KUKA KRL program: ps_a_stb_res_co3.src, ps_a_stb_res_co3.dat

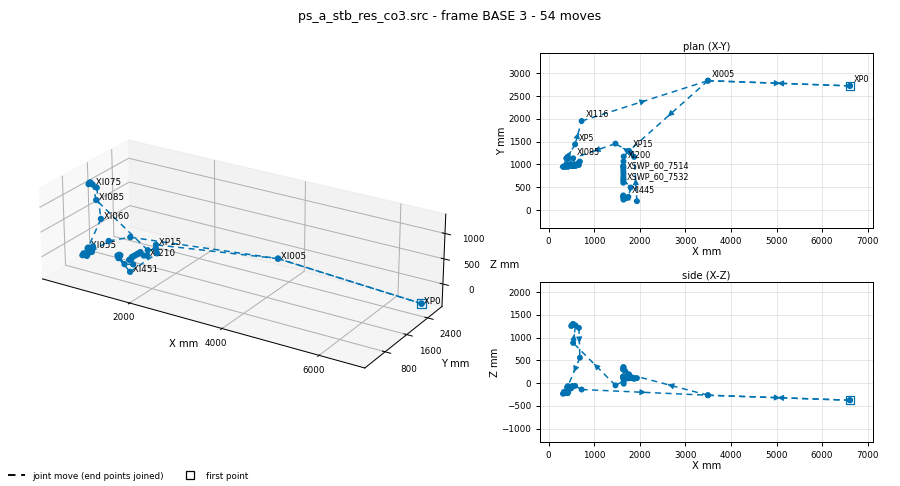
[picture p0: tool path of ps_a_stb_res_co3.src in frame BASE 3, 54 of 54 moves have a stored position in this frame; points joined in program order, loops and branches not executed]
--- ps_a_stb_res_co3.src ---
&ACCESS RVO1
&COMMENT Solda Atego ETB
&PARAM DISKPATH = KRC:\R1\Program\inpro_nao_mexer
DEF ps_a_stb_res_co3( )
;FOLD INI
;FOLD SPOTTECH INI
USERSPOT(#INIT)
;ENDFOLD (SPOTTECH INI)
;FOLD GRIPPERTECH INI
USER_GRP(0,DUMMY,DUMMY,GDEFAULT)
;ENDFOLD (GRIPPERTECH INI)
  ;FOLD USER INI
    ;Make your modifications here

  ;ENDFOLD (USER INI)
;ENDFOLD (INI)

; Caracterizacao dos meios de producao
; Changes: Solda Respot - ATEGO STB
; Versao Atual:05/01/2016
; Ferramenta: Gun C3
; Name: P13.050-R2
; optimised

chk_w4_wechs_ok( )      ; CHECK GUN C3

;FOLD PTP P0 Vel=100 % PDAT0 Tool[4]:Gun C3 Base[3]:Atego/Axor;%{PE}%R 8.2.20,%MKUKATPBASIS,%CMOVE,%VPTP,%P 1:PTP, 2:P0, 3:, 5:100, 7:PDAT0
$BWDSTART=FALSE
PDAT_ACT=PPDAT0
FDAT_ACT=FP0
BAS(#PTP_PARAMS,100)
PTP XP0
;ENDFOLD

if MaxStandMenge (3) then
 MaxStandmengeErreicht (3)
endif

IF (NOT(GHOST())) THEN
if FraesAnf (3) then
 e_fraes4 ( )
endif
ENDIF

;FOLD PTP l005 Vel=100 % P_OLP2 Tool[4]:Gun C3 Base[3]:Atego/Axor;%{PE}%R 8.2.20,%MKUKATPBASIS,%CMOVE,%VPTP,%P 1:PTP, 2:l005, 3:, 5:100, 7:P_OLP2
$BWDSTART=FALSE
PDAT_ACT=PP_OLP2
FDAT_ACT=Fl005
BAS(#PTP_PARAMS,100)
PTP Xl005
;ENDFOLD

; AGUARDA LIBERACAO PARA SOLDAR RESPOT
;FOLD OUT 3338 'R2 solda geometria Ok' State=FALSE ;%{PE}%R 8.2.20,%MKUKATPBASIS,%COUT,%VOUTX,%P 2:3338, 3:R2 solda geometria Ok, 5:FALSE, 6:
$OUT[3338]=FALSE
;ENDFOLD
;FOLD OUT 3348 'Fora area GEOBOX' State=FALSE ;%{PE}%R 8.2.20,%MKUKATPBASIS,%COUT,%VOUTX,%P 2:3348, 3:Fora area GEOBOX, 5:FALSE, 6:
$OUT[3348]=FALSE
;ENDFOLD
;FOLD OUT 3380 'Lib. p/ soldar Res Axor/Atego' State=TRUE ;%{PE}%R 8.2.20,%MKUKATPBASIS,%COUT,%VOUTX,%P 2:3380, 3:Lib. p/ soldar Res Axor/Atego, 5:TRUE, 6:
$OUT[3380]=TRUE
;ENDFOLD
;FOLD WAIT FOR ( IN 3380 'Lib. p/ soldar Res Axor/Atego' );%{PE}%R 8.2.20,%MKUKATPBASIS,%CEXT_WAIT_FOR,%VEXT_WAIT_FOR,%P 2:, 4:, 5:$IN, 6:3380, 7:Lib. p/ soldar Res Axor/Atego, 9:
WAIT FOR  ( $IN[3380] )
;ENDFOLD
;FOLD OUT 3380 'Lib. p/ soldar Res Axor/Atego' State=FALSE ;%{PE}%R 8.2.20,%MKUKATPBASIS,%COUT,%VOUTX,%P 2:3380, 3:Lib. p/ soldar Res Axor/Atego, 5:FALSE, 6:
$OUT[3380]=FALSE
;ENDFOLD

; LIGA INTERTRAVAMENTO 1 C/ R1
;FOLD Collision.Monitoring_1_On ;%{PE}%MKUKATPUSER
COLLSTOP( 1, 1 ) ;Interrupt-Controlled
;ENDFOLD

; LIGA INTERTRAVAMENTO 4 C/ R4
;FOLD Collision.Monitoring_4_On ;%{PE}%MKUKATPUSER
COLLSTOP( 4, 1 ) ;Interrupt-Controlled
;ENDFOLD

; LIGA INTERTRAVAMENTO 12 C/ R1
;FOLD Collision.Monitoring_AREA_6_On ;%{PE}%MKUKATPUSER
COLLSTOP( 12, 1 ) ;not Interrupt-Controlled
;ENDFOLD

;FOLD PTP P15 CONT Vel=100 % xlarge Tool[4]:Gun C3 Base[3]:Atego/Axor;%{PE}%R 8.2.20,%MKUKATPBASIS,%CMOVE,%VPTP,%P 1:PTP, 2:P15, 3:C_DIS, 5:100, 7:xlarge
$BWDSTART=FALSE
PDAT_ACT=Pxlarge
FDAT_ACT=FP15
BAS(#PTP_PARAMS,100)
PTP XP15 C_DIS
;ENDFOLD
;FOLD PTP l210 CONT Vel=100 % large Tool[4]:Gun C3 Base[3]:Atego/Axor;%{PE}%R 8.2.20,%MKUKATPBASIS,%CMOVE,%VPTP,%P 1:PTP, 2:l210, 3:C_DIS, 5:100, 7:large
$BWDSTART=FALSE
PDAT_ACT=Plarge
FDAT_ACT=Fl210
BAS(#PTP_PARAMS,100)
PTP Xl210 C_DIS
;ENDFOLD
;FOLD PTP l200 CONT Vel=100 % medium Tool[4]:Gun C3 Base[3]:Atego/Axor;%{PE}%R 8.2.20,%MKUKATPBASIS,%CMOVE,%VPTP,%P 1:PTP, 2:l200, 3:C_DIS, 5:100, 7:medium
$BWDSTART=FALSE
PDAT_ACT=Pmedium
FDAT_ACT=Fl200
BAS(#PTP_PARAMS,100)
PTP Xl200 C_DIS
;ENDFOLD
;FOLD PTP l195 CONT Vel=100 % fin Tool[4]:Gun C3 Base[3]:Atego/Axor;%{PE}%R 8.2.20,%MKUKATPBASIS,%CMOVE,%VPTP,%P 1:PTP, 2:l195, 3:C_DIS, 5:100, 7:fin
$BWDSTART=FALSE
PDAT_ACT=Pfin
FDAT_ACT=Fl195
BAS(#PTP_PARAMS,100)
PTP Xl195 C_DIS
;ENDFOLD

;FOLD ; SWP_60_7512;%{PE}%R 8.2.20,%MKUKATPBASIS,%CCOMMENT,%VNORMAL,%P 2:SWP_60_7512
;ENDFOLD
;FOLD PTP SWP_60_7512 vmax SPOT Gun=3 RETR CLS PgNo1=204 ACTIVE=1 Tool[4]:Gun C3 Base[3]:Atego/Axor;%{PE}%R 8.2.2,%MKUKATPSPOT,%CSPOT,%VPTP,%P 1:PTP, 2:SWP_60_7512, 3:, 5:100, 7:vmax, 10:3, 12:#FIRST, 14:#CLO, 16:204, 18:1, 20:0, 22:0, 24:1, 25:NORMAL
$BWDSTART=FALSE
PDAT_ACT=Pvmax
FDAT_ACT=FSWP_60_7512
BAS(#PTP_PARAMS,Pvmax.VEL)
S_ACT.GUN=3
S_ACT.PAIR=SDEFAULT.PAIR
S_ACT.RETR=#CLO
S_ACT.CLO_TM=1
S_ACT.PGNO1=204
S_ACT.PGNO2=SDEFAULT.PGNO2
S_ACT.PRESS1=SDEFAULT.PRESS1
S_ACT.PRESS2=SDEFAULT.PRESS2
S_READY=FALSE
PTP XSWP_60_7512
USERSPOT(#SPOT, S_ACT)
WAIT FOR S_READY
;ENDFOLD

;FOLD ; SWP_60_7510;%{PE}%R 8.2.20,%MKUKATPBASIS,%CCOMMENT,%VNORMAL,%P 2:SWP_60_7510
;ENDFOLD
;FOLD PTP SWP_60_7510 vmax SPOT Gun=3 RETR CLS PgNo1=204 ACTIVE=1 Tool[4]:Gun C3 Base[3]:Atego/Axor;%{PE}%R 8.2.2,%MKUKATPSPOT,%CSPOT,%VPTP,%P 1:PTP, 2:SWP_60_7510, 3:, 5:100, 7:vmax, 10:3, 12:#FIRST, 14:#CLO, 16:204, 18:1, 20:0, 22:0, 24:1, 25:NORMAL
$BWDSTART=FALSE
PDAT_ACT=Pvmax
FDAT_ACT=FSWP_60_7510
BAS(#PTP_PARAMS,Pvmax.VEL)
S_ACT.GUN=3
S_ACT.PAIR=SDEFAULT.PAIR
S_ACT.RETR=#CLO
S_ACT.CLO_TM=1
S_ACT.PGNO1=204
S_ACT.PGNO2=SDEFAULT.PGNO2
S_ACT.PRESS1=SDEFAULT.PRESS1
S_ACT.PRESS2=SDEFAULT.PRESS2
S_READY=FALSE
PTP XSWP_60_7510
USERSPOT(#SPOT, S_ACT)
WAIT FOR S_READY
;ENDFOLD

;FOLD ; SWP_60_7508;%{PE}%R 8.2.20,%MKUKATPBASIS,%CCOMMENT,%VNORMAL,%P 2:SWP_60_7508
;ENDFOLD
;FOLD PTP SWP_60_7508 vmax SPOT Gun=3 RETR CLS PgNo1=204 ACTIVE=1 Tool[4]:Gun C3 Base[3]:Atego/Axor;%{PE}%R 8.2.2,%MKUKATPSPOT,%CSPOT,%VPTP,%P 1:PTP, 2:SWP_60_7508, 3:, 5:100, 7:vmax, 10:3, 12:#FIRST, 14:#CLO, 16:204, 18:1, 20:0, 22:0, 24:1, 25:NORMAL
$BWDSTART=FALSE
PDAT_ACT=Pvmax
FDAT_ACT=FSWP_60_7508
BAS(#PTP_PARAMS,Pvmax.VEL)
S_ACT.GUN=3
S_ACT.PAIR=SDEFAULT.PAIR
S_ACT.RETR=#CLO
S_ACT.CLO_TM=1
S_ACT.PGNO1=204
S_ACT.PGNO2=SDEFAULT.PGNO2
S_ACT.PRESS1=SDEFAULT.PRESS1
S_ACT.PRESS2=SDEFAULT.PRESS2
S_READY=FALSE
PTP XSWP_60_7508
USERSPOT(#SPOT, S_ACT)
WAIT FOR S_READY
;ENDFOLD

;FOLD ; SWP_60_7514;%{PE}%R 8.2.20,%MKUKATPBASIS,%CCOMMENT,%VNORMAL,%P 2:SWP_60_7514
;ENDFOLD
;FOLD PTP SWP_60_7514 vmax SPOT Gun=3 RETR CLS PgNo1=204 ACTIVE=1 Tool[4]:Gun C3 Base[3]:Atego/Axor;%{PE}%R 8.2.2,%MKUKATPSPOT,%CSPOT,%VPTP,%P 1:PTP, 2:SWP_60_7514, 3:, 5:100, 7:vmax, 10:3, 12:#FIRST, 14:#CLO, 16:204, 18:1, 20:0, 22:0, 24:1, 25:NORMAL
$BWDSTART=FALSE
PDAT_ACT=Pvmax
FDAT_ACT=FSWP_60_7514
BAS(#PTP_PARAMS,Pvmax.VEL)
S_ACT.GUN=3
S_ACT.PAIR=SDEFAULT.PAIR
S_ACT.RETR=#CLO
S_ACT.CLO_TM=1
S_ACT.PGNO1=204
S_ACT.PGNO2=SDEFAULT.PGNO2
S_ACT.PRESS1=SDEFAULT.PRESS1
S_ACT.PRESS2=SDEFAULT.PRESS2
S_READY=FALSE
PTP XSWP_60_7514
USERSPOT(#SPOT, S_ACT)
WAIT FOR S_READY
;ENDFOLD

;FOLD ; SWP_60_7518;%{PE}%R 8.2.20,%MKUKATPBASIS,%CCOMMENT,%VNORMAL,%P 2:SWP_60_7518
;ENDFOLD
;FOLD PTP SWP_60_7518 vmax SPOT Gun=3 RETR CLS PgNo1=204 ACTIVE=1 Tool[4]:Gun C3 Base[3]:Atego/Axor;%{PE}%R 8.2.2,%MKUKATPSPOT,%CSPOT,%VPTP,%P 1:PTP, 2:SWP_60_7518, 3:, 5:100, 7:vmax, 10:3, 12:#FIRST, 14:#CLO, 16:204, 18:1, 20:0, 22:0, 24:1, 25:NORMAL
$BWDSTART=FALSE
PDAT_ACT=Pvmax
FDAT_ACT=FSWP_60_7518
BAS(#PTP_PARAMS,Pvmax.VEL)
S_ACT.GUN=3
S_ACT.PAIR=SDEFAULT.PAIR
S_ACT.RETR=#CLO
S_ACT.CLO_TM=1
S_ACT.PGNO1=204
S_ACT.PGNO2=SDEFAULT.PGNO2
S_ACT.PRESS1=SDEFAULT.PRESS1
S_ACT.PRESS2=SDEFAULT.PRESS2
S_READY=FALSE
PTP XSWP_60_7518
USERSPOT(#SPOT, S_ACT)
WAIT FOR S_READY
;ENDFOLD

;FOLD ; SWP_60_7522;%{PE}%R 8.2.20,%MKUKATPBASIS,%CCOMMENT,%VNORMAL,%P 2:SWP_60_7522
;ENDFOLD
;FOLD PTP SWP_60_7522 vmax SPOT Gun=3 RETR CLS PgNo1=204 ACTIVE=1 Tool[4]:Gun C3 Base[3]:Atego/Axor;%{PE}%R 8.2.2,%MKUKATPSPOT,%CSPOT,%VPTP,%P 1:PTP, 2:SWP_60_7522, 3:, 5:100, 7:vmax, 10:3, 12:#FIRST, 14:#CLO, 16:204, 18:1, 20:0, 22:0, 24:1, 25:NORMAL
$BWDSTART=FALSE
PDAT_ACT=Pvmax
FDAT_ACT=FSWP_60_7522
BAS(#PTP_PARAMS,Pvmax.VEL)
S_ACT.GUN=3
S_ACT.PAIR=SDEFAULT.PAIR
S_ACT.RETR=#CLO
S_ACT.CLO_TM=1
S_ACT.PGNO1=204
S_ACT.PGNO2=SDEFAULT.PGNO2
S_ACT.PRESS1=SDEFAULT.PRESS1
S_ACT.PRESS2=SDEFAULT.PRESS2
S_READY=FALSE
PTP XSWP_60_7522
USERSPOT(#SPOT, S_ACT)
WAIT FOR S_READY
;ENDFOLD

;FOLD ; SWP_60_7524;%{PE}%R 8.2.20,%MKUKATPBASIS,%CCOMMENT,%VNORMAL,%P 2:SWP_60_7524
;ENDFOLD
;FOLD PTP SWP_60_7524 vmax SPOT Gun=3 RETR CLS PgNo1=204 ACTIVE=1 Tool[4]:Gun C3 Base[3]:Atego/Axor;%{PE}%R 8.2.2,%MKUKATPSPOT,%CSPOT,%VPTP,%P 1:PTP, 2:SWP_60_7524, 3:, 5:100, 7:vmax, 10:3, 12:#FIRST, 14:#CLO, 16:204, 18:1, 20:0, 22:0, 24:1, 25:NORMAL
$BWDSTART=FALSE
PDAT_ACT=Pvmax
FDAT_ACT=FSWP_60_7524
BAS(#PTP_PARAMS,Pvmax.VEL)
S_ACT.GUN=3
S_ACT.PAIR=SDEFAULT.PAIR
S_ACT.RETR=#CLO
S_ACT.CLO_TM=1
S_ACT.PGNO1=204
S_ACT.PGNO2=SDEFAULT.PGNO2
S_ACT.PRESS1=SDEFAULT.PRESS1
S_ACT.PRESS2=SDEFAULT.PRESS2
S_READY=FALSE
PTP XSWP_60_7524
USERSPOT(#SPOT, S_ACT)
WAIT FOR S_READY
;ENDFOLD

;FOLD ; SWP_60_7532;%{PE}%R 8.2.20,%MKUKATPBASIS,%CCOMMENT,%VNORMAL,%P 2:SWP_60_7532
;ENDFOLD
;FOLD PTP SWP_60_7532 vmax SPOT Gun=3 RETR CLS PgNo1=204 ACTIVE=1 Tool[4]:Gun C3 Base[3]:Atego/Axor;%{PE}%R 8.2.2,%MKUKATPSPOT,%CSPOT,%VPTP,%P 1:PTP, 2:SWP_60_7532, 3:, 5:100, 7:vmax, 10:3, 12:#FIRST, 14:#CLO, 16:204, 18:1, 20:0, 22:0, 24:1, 25:NORMAL
$BWDSTART=FALSE
PDAT_ACT=Pvmax
FDAT_ACT=FSWP_60_7532
BAS(#PTP_PARAMS,Pvmax.VEL)
S_ACT.GUN=3
S_ACT.PAIR=SDEFAULT.PAIR
S_ACT.RETR=#CLO
S_ACT.CLO_TM=1
S_ACT.PGNO1=204
S_ACT.PGNO2=SDEFAULT.PGNO2
S_ACT.PRESS1=SDEFAULT.PRESS1
S_ACT.PRESS2=SDEFAULT.PRESS2
S_READY=FALSE
PTP XSWP_60_7532
USERSPOT(#SPOT, S_ACT)
WAIT FOR S_READY
;ENDFOLD

;FOLD PTP l100 CONT Vel=100 % fin Tool[4]:Gun C3 Base[3]:Atego/Axor;%{PE}%R 8.2.20,%MKUKATPBASIS,%CMOVE,%VPTP,%P 1:PTP, 2:l100, 3:C_DIS, 5:100, 7:fin
$BWDSTART=FALSE
PDAT_ACT=Pfin
FDAT_ACT=Fl100
BAS(#PTP_PARAMS,100)
PTP Xl100 C_DIS
;ENDFOLD
;FOLD PTP l101 CONT Vel=100 % small Tool[4]:Gun C3 Base[3]:Atego/Axor;%{PE}%R 8.2.20,%MKUKATPBASIS,%CMOVE,%VPTP,%P 1:PTP, 2:l101, 3:C_DIS, 5:100, 7:small
$BWDSTART=FALSE
PDAT_ACT=Psmall
FDAT_ACT=Fl101
BAS(#PTP_PARAMS,100)
PTP Xl101 C_DIS
;ENDFOLD
;FOLD PTP l445 CONT Vel=100 % small Tool[4]:Gun C3 Base[3]:Atego/Axor;%{PE}%R 8.2.20,%MKUKATPBASIS,%CMOVE,%VPTP,%P 1:PTP, 2:l445, 3:C_DIS, 5:100, 7:small
$BWDSTART=FALSE
PDAT_ACT=Psmall
FDAT_ACT=Fl445
BAS(#PTP_PARAMS,100)
PTP Xl445 C_DIS
;ENDFOLD
;FOLD PTP l446 CONT Vel=100 % fin Tool[4]:Gun C3 Base[3]:Atego/Axor;%{PE}%R 8.2.20,%MKUKATPBASIS,%CMOVE,%VPTP,%P 1:PTP, 2:l446, 3:C_DIS, 5:100, 7:fin
$BWDSTART=FALSE
PDAT_ACT=Pfin
FDAT_ACT=Fl446
BAS(#PTP_PARAMS,100)
PTP Xl446 C_DIS
;ENDFOLD

;FOLD ; SWP_60_7536;%{PE}%R 8.2.20,%MKUKATPBASIS,%CCOMMENT,%VNORMAL,%P 2:SWP_60_7536
;ENDFOLD
;FOLD PTP SWP_60_7537 vmax SPOT Gun=3 RETR CLS PgNo1=204 ACTIVE=1 Tool[4]:Gun C3 Base[3]:Atego/Axor;%{PE}%R 8.2.2,%MKUKATPSPOT,%CSPOT,%VPTP,%P 1:PTP, 2:SWP_60_7537, 3:, 5:100, 7:vmax, 10:3, 12:#FIRST, 14:#CLO, 16:204, 18:1, 20:0, 22:0, 24:1, 25:NORMAL
$BWDSTART=FALSE
PDAT_ACT=Pvmax
FDAT_ACT=FSWP_60_7537
BAS(#PTP_PARAMS,Pvmax.VEL)
S_ACT.GUN=3
S_ACT.PAIR=SDEFAULT.PAIR
S_ACT.RETR=#CLO
S_ACT.CLO_TM=1
S_ACT.PGNO1=204
S_ACT.PGNO2=SDEFAULT.PGNO2
S_ACT.PRESS1=SDEFAULT.PRESS1
S_ACT.PRESS2=SDEFAULT.PRESS2
S_READY=FALSE
PTP XSWP_60_7537
USERSPOT(#SPOT, S_ACT)
WAIT FOR S_READY
;ENDFOLD

;FOLD ; SWP_60_7538;%{PE}%R 8.2.20,%MKUKATPBASIS,%CCOMMENT,%VNORMAL,%P 2:SWP_60_7538
;ENDFOLD
;FOLD PTP SWP_60_7538 vmax SPOT Gun=3 RETR CLS PgNo1=204 ACTIVE=1 Tool[4]:Gun C3 Base[3]:Atego/Axor;%{PE}%R 8.2.2,%MKUKATPSPOT,%CSPOT,%VPTP,%P 1:PTP, 2:SWP_60_7538, 3:, 5:100, 7:vmax, 10:3, 12:#FIRST, 14:#CLO, 16:204, 18:1, 20:0, 22:0, 24:1, 25:NORMAL
$BWDSTART=FALSE
PDAT_ACT=Pvmax
FDAT_ACT=FSWP_60_7538
BAS(#PTP_PARAMS,Pvmax.VEL)
S_ACT.GUN=3
S_ACT.PAIR=SDEFAULT.PAIR
S_ACT.RETR=#CLO
S_ACT.CLO_TM=1
S_ACT.PGNO1=204
S_ACT.PGNO2=SDEFAULT.PGNO2
S_ACT.PRESS1=SDEFAULT.PRESS1
S_ACT.PRESS2=SDEFAULT.PRESS2
S_READY=FALSE
PTP XSWP_60_7538
USERSPOT(#SPOT, S_ACT)
WAIT FOR S_READY
;ENDFOLD

;FOLD ; SWP_60_7540;%{PE}%R 8.2.20,%MKUKATPBASIS,%CCOMMENT,%VNORMAL,%P 2:SWP_60_7540
;ENDFOLD
;FOLD PTP SWP_60_7540 vmax SPOT Gun=3 RETR CLS PgNo1=204 ACTIVE=1 Tool[4]:Gun C3 Base[3]:Atego/Axor;%{PE}%R 8.2.2,%MKUKATPSPOT,%CSPOT,%VPTP,%P 1:PTP, 2:SWP_60_7540, 3:, 5:100, 7:vmax, 10:3, 12:#FIRST, 14:#CLO, 16:204, 18:1, 20:0, 22:0, 24:1, 25:NORMAL
$BWDSTART=FALSE
PDAT_ACT=Pvmax
FDAT_ACT=FSWP_60_7540
BAS(#PTP_PARAMS,Pvmax.VEL)
S_ACT.GUN=3
S_ACT.PAIR=SDEFAULT.PAIR
S_ACT.RETR=#CLO
S_ACT.CLO_TM=1
S_ACT.PGNO1=204
S_ACT.PGNO2=SDEFAULT.PGNO2
S_ACT.PRESS1=SDEFAULT.PRESS1
S_ACT.PRESS2=SDEFAULT.PRESS2
S_READY=FALSE
PTP XSWP_60_7540
USERSPOT(#SPOT, S_ACT)
WAIT FOR S_READY
;ENDFOLD

; LIGA INTERTRAVAMENTO 14 C/ R5
;FOLD Collision.Monitoring_AREA_8_On ;%{PE}%MKUKATPUSER
COLLSTOP( 14, 1 ) ;not Interrupt-Controlled
;ENDFOLD

;FOLD PTP l447 CONT Vel=100 % fin Tool[4]:Gun C3 Base[3]:Atego/Axor;%{PE}%R 8.2.20,%MKUKATPBASIS,%CMOVE,%VPTP,%P 1:PTP, 2:l447, 3:C_DIS, 5:100, 7:fin
$BWDSTART=FALSE
PDAT_ACT=Pfin
FDAT_ACT=Fl447
BAS(#PTP_PARAMS,100)
PTP Xl447 C_DIS
;ENDFOLD
;FOLD PTP l451 CONT Vel=100 % medium Tool[4]:Gun C3 Base[3]:Atego/Axor;%{PE}%R 8.2.20,%MKUKATPBASIS,%CMOVE,%VPTP,%P 1:PTP, 2:l451, 3:C_DIS, 5:100, 7:medium
$BWDSTART=FALSE
PDAT_ACT=Pmedium
FDAT_ACT=Fl451
BAS(#PTP_PARAMS,100)
PTP Xl451 C_DIS
;ENDFOLD
;FOLD PTP l103 CONT Vel=100 % medium Tool[4]:Gun C3 Base[3]:Atego/Axor;%{PE}%R 8.2.20,%MKUKATPBASIS,%CMOVE,%VPTP,%P 1:PTP, 2:l103, 3:C_DIS, 5:100, 7:medium
$BWDSTART=FALSE
PDAT_ACT=Pmedium
FDAT_ACT=Fl103
BAS(#PTP_PARAMS,100)
PTP Xl103 C_DIS
;ENDFOLD
;FOLD PTP l090 CONT Vel=100 % xlarge Tool[4]:Gun C3 Base[3]:Atego/Axor;%{PE}%R 8.2.20,%MKUKATPBASIS,%CMOVE,%VPTP,%P 1:PTP, 2:l090, 3:C_DIS, 5:100, 7:xlarge
$BWDSTART=FALSE
PDAT_ACT=Pxlarge
FDAT_ACT=Fl090
BAS(#PTP_PARAMS,100)
PTP Xl090 C_DIS
;ENDFOLD
;FOLD PTP l091 CONT Vel=100 % xlarge Tool[4]:Gun C3 Base[3]:Atego/Axor;%{PE}%R 8.2.20,%MKUKATPBASIS,%CMOVE,%VPTP,%P 1:PTP, 2:l091, 3:C_DIS, 5:100, 7:xlarge
$BWDSTART=FALSE
PDAT_ACT=Pxlarge
FDAT_ACT=Fl091
BAS(#PTP_PARAMS,100)
PTP Xl091 C_DIS
;ENDFOLD
;FOLD PTP l085 CONT Vel=100 % large Tool[4]:Gun C3 Base[3]:Atego/Axor;%{PE}%R 8.2.20,%MKUKATPBASIS,%CMOVE,%VPTP,%P 1:PTP, 2:l085, 3:C_DIS, 5:100, 7:large
$BWDSTART=FALSE
PDAT_ACT=Plarge
FDAT_ACT=Fl085
BAS(#PTP_PARAMS,100)
PTP Xl085 C_DIS
;ENDFOLD
;FOLD PTP l075 CONT Vel=100 % fin Tool[4]:Gun C3 Base[3]:Atego/Axor;%{PE}%R 8.2.20,%MKUKATPBASIS,%CMOVE,%VPTP,%P 1:PTP, 2:l075, 3:C_DIS, 5:100, 7:fin
$BWDSTART=FALSE
PDAT_ACT=Pfin
FDAT_ACT=Fl075
BAS(#PTP_PARAMS,100)
PTP Xl075 C_DIS
;ENDFOLD

;FOLD ; SWP_60_7784;%{PE}%R 8.2.20,%MKUKATPBASIS,%CCOMMENT,%VNORMAL,%P 2:SWP_60_7784
;ENDFOLD
;FOLD PTP SWP_60_7784 vmax SPOT Gun=3 RETR CLS PgNo1=201 ACTIVE=1 Tool[4]:Gun C3 Base[3]:Atego/Axor;%{PE}%R 8.2.2,%MKUKATPSPOT,%CSPOT,%VPTP,%P 1:PTP, 2:SWP_60_7784, 3:, 5:100, 7:vmax, 10:3, 12:#FIRST, 14:#CLO, 16:201, 18:1, 20:0, 22:0, 24:1, 25:NORMAL
$BWDSTART=FALSE
PDAT_ACT=Pvmax
FDAT_ACT=FSWP_60_7784
BAS(#PTP_PARAMS,Pvmax.VEL)
S_ACT.GUN=3
S_ACT.PAIR=SDEFAULT.PAIR
S_ACT.RETR=#CLO
S_ACT.CLO_TM=1
S_ACT.PGNO1=201
S_ACT.PGNO2=SDEFAULT.PGNO2
S_ACT.PRESS1=SDEFAULT.PRESS1
S_ACT.PRESS2=SDEFAULT.PRESS2
S_READY=FALSE
PTP XSWP_60_7784
USERSPOT(#SPOT, S_ACT)
WAIT FOR S_READY
;ENDFOLD

; DESLIGA INTERTRAVAMENTO 12 C/ R1
;FOLD Collision.Monitoring_AREA_6_Off . ;%{PE}%MKUKATPUSER
COLLSTOP( 12, 2+0 )
;ENDFOLD

;FOLD ; SWP_60_7782;%{PE}%R 8.2.20,%MKUKATPBASIS,%CCOMMENT,%VNORMAL,%P 2:SWP_60_7782
;ENDFOLD
;FOLD PTP SWP_60_7782 vmax SPOT Gun=3 RETR CLS PgNo1=201 ACTIVE=1 Tool[4]:Gun C3 Base[3]:Atego/Axor;%{PE}%R 8.2.2,%MKUKATPSPOT,%CSPOT,%VPTP,%P 1:PTP, 2:SWP_60_7782, 3:, 5:100, 7:vmax, 10:3, 12:#FIRST, 14:#CLO, 16:201, 18:1, 20:0, 22:0, 24:1, 25:NORMAL
$BWDSTART=FALSE
PDAT_ACT=Pvmax
FDAT_ACT=FSWP_60_7782
BAS(#PTP_PARAMS,Pvmax.VEL)
S_ACT.GUN=3
S_ACT.PAIR=SDEFAULT.PAIR
S_ACT.RETR=#CLO
S_ACT.CLO_TM=1
S_ACT.PGNO1=201
S_ACT.PGNO2=SDEFAULT.PGNO2
S_ACT.PRESS1=SDEFAULT.PRESS1
S_ACT.PRESS2=SDEFAULT.PRESS2
S_READY=FALSE
PTP XSWP_60_7782
USERSPOT(#SPOT, S_ACT)
WAIT FOR S_READY
;ENDFOLD

;FOLD ; SWP_60_7780;%{PE}%R 8.2.20,%MKUKATPBASIS,%CCOMMENT,%VNORMAL,%P 2:SWP_60_7780
;ENDFOLD
;FOLD PTP SWP_60_7780 vmax SPOT Gun=3 RETR CLS PgNo1=201 ACTIVE=1 Tool[4]:Gun C3 Base[3]:Atego/Axor;%{PE}%R 8.2.2,%MKUKATPSPOT,%CSPOT,%VPTP,%P 1:PTP, 2:SWP_60_7780, 3:, 5:100, 7:vmax, 10:3, 12:#FIRST, 14:#CLO, 16:201, 18:1, 20:0, 22:0, 24:1, 25:NORMAL
$BWDSTART=FALSE
PDAT_ACT=Pvmax
FDAT_ACT=FSWP_60_7780
BAS(#PTP_PARAMS,Pvmax.VEL)
S_ACT.GUN=3
S_ACT.PAIR=SDEFAULT.PAIR
S_ACT.RETR=#CLO
S_ACT.CLO_TM=1
S_ACT.PGNO1=201
S_ACT.PGNO2=SDEFAULT.PGNO2
S_ACT.PRESS1=SDEFAULT.PRESS1
S_ACT.PRESS2=SDEFAULT.PRESS2
S_READY=FALSE
PTP XSWP_60_7780
USERSPOT(#SPOT, S_ACT)
WAIT FOR S_READY
;ENDFOLD

;FOLD PTP l070 CONT Vel=100 % small Tool[4]:Gun C3 Base[3]:Atego/Axor;%{PE}%R 8.2.20,%MKUKATPBASIS,%CMOVE,%VPTP,%P 1:PTP, 2:l070, 3:C_DIS, 5:100, 7:small
$BWDSTART=FALSE
PDAT_ACT=Psmall
FDAT_ACT=Fl070
BAS(#PTP_PARAMS,100)
PTP Xl070 C_DIS
;ENDFOLD
;FOLD PTP l060 Vel=100 % P_OLP13 Tool[4]:Gun C3 Base[3]:Atego/Axor;%{PE}%R 8.2.20,%MKUKATPBASIS,%CMOVE,%VPTP,%P 1:PTP, 2:l060, 3:, 5:100, 7:P_OLP13
$BWDSTART=FALSE
PDAT_ACT=PP_OLP13
FDAT_ACT=Fl060
BAS(#PTP_PARAMS,100)
PTP Xl060
;ENDFOLD

; DESLIGA INTERTRAVAMENTO 14 C/ R5
;FOLD Collision.Monitoring_AREA_8_Off . ;%{PE}%MKUKATPUSER
COLLSTOP( 14, 2+0 )
;ENDFOLD

; LIGA INTERTRAVAMENTO 13 C/ R5
;FOLD Collision.Monitoring_AREA_7_On ;%{PE}%MKUKATPUSER
COLLSTOP( 13, 1 ) ;not Interrupt-Controlled
;ENDFOLD

;FOLD PTP l055 CONT Vel=100 % fin Tool[4]:Gun C3 Base[3]:Atego/Axor;%{PE}%R 8.2.20,%MKUKATPBASIS,%CMOVE,%VPTP,%P 1:PTP, 2:l055, 3:C_DIS, 5:100, 7:fin
$BWDSTART=FALSE
PDAT_ACT=Pfin
FDAT_ACT=Fl055
BAS(#PTP_PARAMS,100)
PTP Xl055 C_DIS
;ENDFOLD

;FOLD ; SWP_60_9076;%{PE}%R 8.2.20,%MKUKATPBASIS,%CCOMMENT,%VNORMAL,%P 2:SWP_60_9076
;ENDFOLD
;FOLD PTP SWP_60_9076 vmax SPOT Gun=3 RETR CLS PgNo1=202 ACTIVE=1 Tool[4]:Gun C3 Base[3]:Atego/Axor;%{PE}%R 8.2.2,%MKUKATPSPOT,%CSPOT,%VPTP,%P 1:PTP, 2:SWP_60_9076, 3:, 5:100, 7:vmax, 10:3, 12:#FIRST, 14:#CLO, 16:202, 18:1, 20:0, 22:0, 24:1, 25:NORMAL
$BWDSTART=FALSE
PDAT_ACT=Pvmax
FDAT_ACT=FSWP_60_9076
BAS(#PTP_PARAMS,Pvmax.VEL)
S_ACT.GUN=3
S_ACT.PAIR=SDEFAULT.PAIR
S_ACT.RETR=#CLO
S_ACT.CLO_TM=1
S_ACT.PGNO1=202
S_ACT.PGNO2=SDEFAULT.PGNO2
S_ACT.PRESS1=SDEFAULT.PRESS1
S_ACT.PRESS2=SDEFAULT.PRESS2
S_READY=FALSE
PTP XSWP_60_9076
USERSPOT(#SPOT, S_ACT)
WAIT FOR S_READY
;ENDFOLD

;FOLD ; SWP_60_9074;%{PE}%R 8.2.20,%MKUKATPBASIS,%CCOMMENT,%VNORMAL,%P 2:SWP_60_9074
;ENDFOLD
;FOLD PTP SWP_60_9074 vmax SPOT Gun=3 RETR CLS PgNo1=202 ACTIVE=1 Tool[4]:Gun C3 Base[3]:Atego/Axor;%{PE}%R 8.2.2,%MKUKATPSPOT,%CSPOT,%VPTP,%P 1:PTP, 2:SWP_60_9074, 3:, 5:100, 7:vmax, 10:3, 12:#FIRST, 14:#CLO, 16:202, 18:1, 20:0, 22:0, 24:1, 25:NORMAL
$BWDSTART=FALSE
PDAT_ACT=Pvmax
FDAT_ACT=FSWP_60_9074
BAS(#PTP_PARAMS,Pvmax.VEL)
S_ACT.GUN=3
S_ACT.PAIR=SDEFAULT.PAIR
S_ACT.RETR=#CLO
S_ACT.CLO_TM=1
S_ACT.PGNO1=202
S_ACT.PGNO2=SDEFAULT.PGNO2
S_ACT.PRESS1=SDEFAULT.PRESS1
S_ACT.PRESS2=SDEFAULT.PRESS2
S_READY=FALSE
PTP XSWP_60_9074
USERSPOT(#SPOT, S_ACT)
WAIT FOR S_READY
;ENDFOLD

;FOLD ; SWP_60_9072;%{PE}%R 8.2.20,%MKUKATPBASIS,%CCOMMENT,%VNORMAL,%P 2:SWP_60_9072
;ENDFOLD
;FOLD PTP SWP_60_9072 vmax SPOT Gun=3 RETR CLS PgNo1=202 ACTIVE=1 Tool[4]:Gun C3 Base[3]:Atego/Axor;%{PE}%R 8.2.2,%MKUKATPSPOT,%CSPOT,%VPTP,%P 1:PTP, 2:SWP_60_9072, 3:, 5:100, 7:vmax, 10:3, 12:#FIRST, 14:#CLO, 16:202, 18:1, 20:0, 22:0, 24:1, 25:NORMAL
$BWDSTART=FALSE
PDAT_ACT=Pvmax
FDAT_ACT=FSWP_60_9072
BAS(#PTP_PARAMS,Pvmax.VEL)
S_ACT.GUN=3
S_ACT.PAIR=SDEFAULT.PAIR
S_ACT.RETR=#CLO
S_ACT.CLO_TM=1
S_ACT.PGNO1=202
S_ACT.PGNO2=SDEFAULT.PGNO2
S_ACT.PRESS1=SDEFAULT.PRESS1
S_ACT.PRESS2=SDEFAULT.PRESS2
S_READY=FALSE
PTP XSWP_60_9072
USERSPOT(#SPOT, S_ACT)
WAIT FOR S_READY
;ENDFOLD

;FOLD ; SWP_60_9070;%{PE}%R 8.2.20,%MKUKATPBASIS,%CCOMMENT,%VNORMAL,%P 2:SWP_60_9070
;ENDFOLD
;FOLD PTP SWP_60_9070 vmax SPOT Gun=3 RETR CLS PgNo1=202 ACTIVE=1 Tool[4]:Gun C3 Base[3]:Atego/Axor;%{PE}%R 8.2.2,%MKUKATPSPOT,%CSPOT,%VPTP,%P 1:PTP, 2:SWP_60_9070, 3:, 5:100, 7:vmax, 10:3, 12:#FIRST, 14:#CLO, 16:202, 18:1, 20:0, 22:0, 24:1, 25:NORMAL
$BWDSTART=FALSE
PDAT_ACT=Pvmax
FDAT_ACT=FSWP_60_9070
BAS(#PTP_PARAMS,Pvmax.VEL)
S_ACT.GUN=3
S_ACT.PAIR=SDEFAULT.PAIR
S_ACT.RETR=#CLO
S_ACT.CLO_TM=1
S_ACT.PGNO1=202
S_ACT.PGNO2=SDEFAULT.PGNO2
S_ACT.PRESS1=SDEFAULT.PRESS1
S_ACT.PRESS2=SDEFAULT.PRESS2
S_READY=FALSE
PTP XSWP_60_9070
USERSPOT(#SPOT, S_ACT)
WAIT FOR S_READY
;ENDFOLD

;FOLD PTP l050 CONT Vel=100 % fin Tool[4]:Gun C3 Base[3]:Atego/Axor;%{PE}%R 8.2.20,%MKUKATPBASIS,%CMOVE,%VPTP,%P 1:PTP, 2:l050, 3:C_DIS, 5:100, 7:fin
$BWDSTART=FALSE
PDAT_ACT=Pfin
FDAT_ACT=Fl050
BAS(#PTP_PARAMS,100)
PTP Xl050 C_DIS
;ENDFOLD
;FOLD PTP l040 CONT Vel=100 % xlarge Tool[4]:Gun C3 Base[3]:Atego/Axor;%{PE}%R 8.2.20,%MKUKATPBASIS,%CMOVE,%VPTP,%P 1:PTP, 2:l040, 3:C_DIS, 5:100, 7:xlarge
$BWDSTART=FALSE
PDAT_ACT=Pxlarge
FDAT_ACT=Fl040
BAS(#PTP_PARAMS,100)
PTP Xl040 C_DIS
;ENDFOLD
;FOLD PTP l035 CONT Vel=100 % medium Tool[4]:Gun C3 Base[3]:Atego/Axor;%{PE}%R 8.2.20,%MKUKATPBASIS,%CMOVE,%VPTP,%P 1:PTP, 2:l035, 3:C_DIS, 5:100, 7:medium
$BWDSTART=FALSE
PDAT_ACT=Pmedium
FDAT_ACT=Fl035
BAS(#PTP_PARAMS,100)
PTP Xl035 C_DIS
;ENDFOLD
;FOLD PTP l025 CONT Vel=100 % fin Tool[4]:Gun C3 Base[3]:Atego/Axor;%{PE}%R 8.2.20,%MKUKATPBASIS,%CMOVE,%VPTP,%P 1:PTP, 2:l025, 3:C_DIS, 5:100, 7:fin
$BWDSTART=FALSE
PDAT_ACT=Pfin
FDAT_ACT=Fl025
BAS(#PTP_PARAMS,100)
PTP Xl025 C_DIS
;ENDFOLD

;FOLD ; SWP_60_9054;%{PE}%R 8.2.20,%MKUKATPBASIS,%CCOMMENT,%VNORMAL,%P 2:SWP_60_9054
;ENDFOLD
;FOLD PTP SWP_60_9054 vmax SPOT Gun=3 RETR CLS PgNo1=203 ACTIVE=1 Tool[4]:Gun C3 Base[3]:Atego/Axor;%{PE}%R 8.2.2,%MKUKATPSPOT,%CSPOT,%VPTP,%P 1:PTP, 2:SWP_60_9054, 3:, 5:100, 7:vmax, 10:3, 12:#FIRST, 14:#CLO, 16:203, 18:1, 20:0, 22:0, 24:1, 25:NORMAL
$BWDSTART=FALSE
PDAT_ACT=Pvmax
FDAT_ACT=FSWP_60_9054
BAS(#PTP_PARAMS,Pvmax.VEL)
S_ACT.GUN=3
S_ACT.PAIR=SDEFAULT.PAIR
S_ACT.RETR=#CLO
S_ACT.CLO_TM=1
S_ACT.PGNO1=203
S_ACT.PGNO2=SDEFAULT.PGNO2
S_ACT.PRESS1=SDEFAULT.PRESS1
S_ACT.PRESS2=SDEFAULT.PRESS2
S_READY=FALSE
PTP XSWP_60_9054
USERSPOT(#SPOT, S_ACT)
WAIT FOR S_READY
;ENDFOLD

;FOLD ; SWP_60_9048;%{PE}%R 8.2.20,%MKUKATPBASIS,%CCOMMENT,%VNORMAL,%P 2:SWP_60_9048
;ENDFOLD
;FOLD PTP SWP_60_9048 vmax SPOT Gun=3 RETR CLS PgNo1=203 ACTIVE=1 Tool[4]:Gun C3 Base[3]:Atego/Axor;%{PE}%R 8.2.2,%MKUKATPSPOT,%CSPOT,%VPTP,%P 1:PTP, 2:SWP_60_9048, 3:, 5:100, 7:vmax, 10:3, 12:#FIRST, 14:#CLO, 16:203, 18:1, 20:0, 22:0, 24:1, 25:NORMAL
$BWDSTART=FALSE
PDAT_ACT=Pvmax
FDAT_ACT=FSWP_60_9048
BAS(#PTP_PARAMS,Pvmax.VEL)
S_ACT.GUN=3
S_ACT.PAIR=SDEFAULT.PAIR
S_ACT.RETR=#CLO
S_ACT.CLO_TM=1
S_ACT.PGNO1=203
S_ACT.PGNO2=SDEFAULT.PGNO2
S_ACT.PRESS1=SDEFAULT.PRESS1
S_ACT.PRESS2=SDEFAULT.PRESS2
S_READY=FALSE
PTP XSWP_60_9048
USERSPOT(#SPOT, S_ACT)
WAIT FOR S_READY
;ENDFOLD

;FOLD ; SWP_60_9050;%{PE}%R 8.2.20,%MKUKATPBASIS,%CCOMMENT,%VNORMAL,%P 2:SWP_60_9050
;ENDFOLD
;FOLD PTP SWP_60_9050 vmax SPOT Gun=3 RETR CLS PgNo1=203 ACTIVE=1 Tool[4]:Gun C3 Base[3]:Atego/Axor;%{PE}%R 8.2.2,%MKUKATPSPOT,%CSPOT,%VPTP,%P 1:PTP, 2:SWP_60_9050, 3:, 5:100, 7:vmax, 10:3, 12:#FIRST, 14:#CLO, 16:203, 18:1, 20:0, 22:0, 24:1, 25:NORMAL
$BWDSTART=FALSE
PDAT_ACT=Pvmax
FDAT_ACT=FSWP_60_9050
BAS(#PTP_PARAMS,Pvmax.VEL)
S_ACT.GUN=3
S_ACT.PAIR=SDEFAULT.PAIR
S_ACT.RETR=#CLO
S_ACT.CLO_TM=1
S_ACT.PGNO1=203
S_ACT.PGNO2=SDEFAULT.PGNO2
S_ACT.PRESS1=SDEFAULT.PRESS1
S_ACT.PRESS2=SDEFAULT.PRESS2
S_READY=FALSE
PTP XSWP_60_9050
USERSPOT(#SPOT, S_ACT)
WAIT FOR S_READY
;ENDFOLD

;FOLD PTP P1 CONT Vel=100 % fin Tool[4]:Gun C3 Base[3]:Atego/Axor;%{PE}%R 8.2.20,%MKUKATPBASIS,%CMOVE,%VPTP,%P 1:PTP, 2:P1, 3:C_DIS, 5:100, 7:fin
$BWDSTART=FALSE
PDAT_ACT=Pfin
FDAT_ACT=FP1
BAS(#PTP_PARAMS,100)
PTP XP1 C_DIS
;ENDFOLD

;FOLD ; SWP_60_9052;%{PE}%R 8.2.20,%MKUKATPBASIS,%CCOMMENT,%VNORMAL,%P 2:SWP_60_9052
;ENDFOLD
;FOLD PTP SWP_60_9052 vmax SPOT Gun=3 RETR CLS PgNo1=203 ACTIVE=1 Tool[4]:Gun C3 Base[3]:Atego/Axor;%{PE}%R 8.2.2,%MKUKATPSPOT,%CSPOT,%VPTP,%P 1:PTP, 2:SWP_60_9052, 3:, 5:100, 7:vmax, 10:3, 12:#FIRST, 14:#CLO, 16:203, 18:1, 20:0, 22:0, 24:1, 25:NORMAL
$BWDSTART=FALSE
PDAT_ACT=Pvmax
FDAT_ACT=FSWP_60_9052
BAS(#PTP_PARAMS,Pvmax.VEL)
S_ACT.GUN=3
S_ACT.PAIR=SDEFAULT.PAIR
S_ACT.RETR=#CLO
S_ACT.CLO_TM=1
S_ACT.PGNO1=203
S_ACT.PGNO2=SDEFAULT.PGNO2
S_ACT.PRESS1=SDEFAULT.PRESS1
S_ACT.PRESS2=SDEFAULT.PRESS2
S_READY=FALSE
PTP XSWP_60_9052
USERSPOT(#SPOT, S_ACT)
WAIT FOR S_READY
;ENDFOLD

;FOLD PTP l020 CONT Vel=100 % fin Tool[4]:Gun C3 Base[3]:Atego/Axor;%{PE}%R 8.2.20,%MKUKATPBASIS,%CMOVE,%VPTP,%P 1:PTP, 2:l020, 3:C_DIS, 5:100, 7:fin
$BWDSTART=FALSE
PDAT_ACT=Pfin
FDAT_ACT=Fl020
BAS(#PTP_PARAMS,100)
PTP Xl020 C_DIS
;ENDFOLD
;FOLD PTP l010 CONT Vel=100 % medium Tool[4]:Gun C3 Base[3]:Atego/Axor;%{PE}%R 8.2.20,%MKUKATPBASIS,%CMOVE,%VPTP,%P 1:PTP, 2:l010, 3:C_DIS, 5:100, 7:medium
$BWDSTART=FALSE
PDAT_ACT=Pmedium
FDAT_ACT=Fl010
BAS(#PTP_PARAMS,100)
PTP Xl010 C_DIS
;ENDFOLD
;FOLD PTP P4 CONT Vel=100 % xlarge Tool[4]:Gun C3 Base[3]:Atego/Axor;%{PE}%R 8.2.20,%MKUKATPBASIS,%CMOVE,%VPTP,%P 1:PTP, 2:P4, 3:C_DIS, 5:100, 7:xlarge
$BWDSTART=FALSE
PDAT_ACT=Pxlarge
FDAT_ACT=FP4
BAS(#PTP_PARAMS,100)
PTP XP4 C_DIS
;ENDFOLD
;FOLD PTP P5 CONT Vel=100 % xlarge Tool[4]:Gun C3 Base[3]:Atego/Axor;%{PE}%R 8.2.20,%MKUKATPBASIS,%CMOVE,%VPTP,%P 1:PTP, 2:P5, 3:C_DIS, 5:100, 7:xlarge
$BWDSTART=FALSE
PDAT_ACT=Pxlarge
FDAT_ACT=FP5
BAS(#PTP_PARAMS,100)
PTP XP5 C_DIS
;ENDFOLD
;FOLD PTP l116 Vel=100 % vmax Tool[4]:Gun C3 Base[3]:Atego/Axor;%{PE}%R 8.2.20,%MKUKATPBASIS,%CMOVE,%VPTP,%P 1:PTP, 2:l116, 3:, 5:100, 7:vmax
$BWDSTART=FALSE
PDAT_ACT=Pvmax
FDAT_ACT=Fl116
BAS(#PTP_PARAMS,100)
PTP Xl116
;ENDFOLD

; DESLIGA INTERTRAVAMENTO 13 C/ R5
;FOLD Collision.Monitoring_AREA_7_Off . ;%{PE}%MKUKATPUSER
COLLSTOP( 13, 2+0 )
;ENDFOLD

; FIM DE TRABALHO RESPOT
;FOLD PULSE 3333 'R2 trabalho concluído' State=TRUE Time=3 sec;%{PE}%R 8.2.20,%MKUKATPBASIS,%COUT,%VPULSE,%P 2:3333, 3:R2 trabalho concluído, 5:TRUE, 6:, 8:3
PULSE($OUT[3333], TRUE,3)
;ENDFOLD
;FOLD OUT 3348 'Fora area GEOBOX' State=TRUE ;%{PE}%R 8.2.20,%MKUKATPBASIS,%COUT,%VOUTX,%P 2:3348, 3:Fora area GEOBOX, 5:TRUE, 6:
$OUT[3348]=TRUE
;ENDFOLD

;FOLD SYN OUT 3340 'AREA_CLEAR_AGV' State=TRUE at START Delay=0 ms;%{PE}%R 8.2.20,%MKUKATPBASIS,%COUT,%VSYNOUT,%P 2:3340, 3:AREA_CLEAR_AGV, 5:TRUE, 7:0, 9:0, 12:0
TRIGGER WHEN DISTANCE=0 DELAY=0 DO $OUT[3340]=TRUE
;ENDFOLD
; DESLIGA INTERTRAVAMENTO 1 C/ R1
;FOLD Collision.Monitoring_1_Off . ;%{PE}%MKUKATPUSER
COLLSTOP( 1, 2+0 )
;ENDFOLD

; DESLIGA INTERTRAVAMENTO 4 C/ R4
;FOLD Collision.Monitoring_4_Off . ;%{PE}%MKUKATPUSER
COLLSTOP( 4, 2+0 )
;ENDFOLD

;FOLD PTP l120 CONT Vel=100 % xxlarge Tool[4]:Gun C3 Base[3]:Atego/Axor;%{PE}%R 8.2.20,%MKUKATPBASIS,%CMOVE,%VPTP,%P 1:PTP, 2:l120, 3:C_DIS, 5:100, 7:xxlarge
$BWDSTART=FALSE
PDAT_ACT=Pxxlarge
FDAT_ACT=Fl120
BAS(#PTP_PARAMS,100)
PTP Xl120 C_DIS
;ENDFOLD
;FOLD PTP P6 Vel=100 % PDAT6 Tool[4]:Gun C3 Base[3]:Atego/Axor;%{PE}%R 8.2.20,%MKUKATPBASIS,%CMOVE,%VPTP,%P 1:PTP, 2:P6, 3:, 5:100, 7:PDAT6
$BWDSTART=FALSE
PDAT_ACT=PPDAT6
FDAT_ACT=FP6
BAS(#PTP_PARAMS,100)
PTP XP6
;ENDFOLD

IF(NOT(GHOST())) THEN
if FraesAnf (3) then
f_fraes4 ()
endif
ENDIF




END

--- ps_a_stb_res_co3.dat ---
&ACCESS RVO1
&COMMENT Solda Atego ETB
&PARAM DISKPATH = KRC:\R1\Program\inpro_nao_mexer
DEFDAT ps_a_stb_res_co3
;FOLD EXTERNAL DECLARATIONS;%{PE}%MKUKATPBASIS,%CEXT,%VCOMMON,%P
;FOLD GRIPPERTECH EXT
EXT  H50 (INT  :IN,INT  :IN,INT  :IN,GRP_TYP  :IN )
;ENDFOLD (GRIPPERTECH EXT)
;FOLD SPOTTECH EXT
EXT  USERSPOT (S_COMMAND  :IN,SPOT_TYPE  :IN )
;ENDFOLD (SPOTTECH EXT)
;FOLD BASISTECH EXT;%{PE}%MKUKATPBASIS,%CEXT,%VEXT,%P
EXT  BAS (BAS_COMMAND  :IN,REAL  :IN )
DECL INT SUCCESS
;ENDFOLD (BASISTECH EXT)
;FOLD USER EXT;%{E}%MKUKATPUSER,%CEXT,%VEXT,%P
;Make your modifications here

;ENDFOLD (USER EXT)
;ENDFOLD (EXTERNAL DECLARATIONS)
DECL FDAT Fl010={TOOL_NO 4,BASE_NO 3,IPO_FRAME #BASE,POINT2[] " "}
DECL PDAT PP_OLP3={VEL 100.0,ACC 100.0,APO_DIST 20.0,APO_MODE #CDIS}
DECL E6POS Xl010={X 392.920105,Y 1131.21802,Z -209.606003,A -17.6636105,B -79.1884537,C -69.3054886,S 2,T 10,E1 -5800.0,E2 0.0,E3 0.0,E4 0.0,E5 0.0,E6 0.0}
DECL FDAT Fl015={TOOL_NO 4,BASE_NO 3,IPO_FRAME #BASE,POINT2[] " "}
DECL PDAT PP_OLP4={VEL 100.0,ACC 100.0,APO_DIST 20.0,APO_MODE #CDIS}
DECL E6POS Xl015={X 337.123596,Y 947.304626,Z -231.1129,A -0.312473506,B -83.5992584,C -88.2265625,S 2,T 11,E1 -5800.0,E2 0.0,E3 0.0,E4 0.0,E5 0.0,E6 0.0}
DECL FDAT Fl020={TOOL_NO 4,BASE_NO 3,IPO_FRAME #BASE,POINT2[] " "}
DECL PDAT PP_OLP5={VEL 100.0,ACC 100.0,APO_DIST 20.0,APO_MODE #CDIS}
DECL E6POS Xl020={X 313.714386,Y 948.87738,Z -230.098694,A -13.2213497,B -83.3848572,C -76.0714264,S 2,T 11,E1 -5800.00098,E2 0.0,E3 0.0,E4 0.0,E5 0.0,E6 0.0}
DECL LDAT LL_OLP1={VEL 2.0,ACC 100.0,APO_DIST 0.0,APO_FAC 0.0,ORI_TYP #VAR,CIRC_TYP #BASE,JERK_FAC 50.0}
DECL LDAT LL_OLP2={VEL 2.0,ACC 100.0,APO_DIST 0.0,APO_FAC 0.0,ORI_TYP #VAR,CIRC_TYP #BASE,JERK_FAC 50.0}
DECL LDAT LL_OLP3={VEL 2.0,ACC 100.0,APO_DIST 0.0,APO_FAC 0.0,ORI_TYP #VAR,CIRC_TYP #BASE,JERK_FAC 50.0}
DECL LDAT LL_OLP4={VEL 2.0,ACC 100.0,APO_DIST 0.0,APO_FAC 0.0,ORI_TYP #VAR,CIRC_TYP #BASE,JERK_FAC 50.0}
DECL FDAT Fl025={TOOL_NO 4,BASE_NO 3,IPO_FRAME #BASE,POINT2[] " "}
DECL PDAT PP_OLP6={VEL 100.0,ACC 100.0,APO_DIST 10.0,APO_MODE #CDIS}
DECL E6POS Xl025={X 419.118195,Y 948.157227,Z -219.959106,A -10.0680199,B -82.4983597,C -78.8929672,S 2,T 11,E1 -5800.0,E2 0.0,E3 0.0,E4 0.0,E5 0.0,E6 0.0}
DECL FDAT Fl030={TOOL_NO 4,BASE_NO 3,IPO_FRAME #BASE,POINT2[] " "}
DECL PDAT PP_OLP7={VEL 100.0,ACC 100.0,APO_DIST 10.0,APO_MODE #CDIS}
DECL E6POS Xl030={X 410.335693,Y 949.091919,Z -235.275803,A 0.560922086,B -77.4818726,C -89.0896072,S 2,T 11,E1 -5800.0,E2 0.0,E3 0.0,E4 0.0,E5 0.0,E6 0.0}
DECL FDAT Fl035={TOOL_NO 4,BASE_NO 3,IPO_FRAME #BASE,POINT2[] " "}
DECL PDAT PP_OLP8={VEL 100.0,ACC 100.0,APO_DIST 10.0,APO_MODE #CDIS}
DECL E6POS Xl035={X 393.480988,Y 1140.57202,Z -217.210007,A -166.776901,B -69.7256012,C 76.8141098,S 2,T 10,E1 -5800.0,E2 0.0,E3 0.0,E4 0.0,E5 0.0,E6 0.0}
DECL FDAT Fl040={TOOL_NO 4,BASE_NO 3,IPO_FRAME #BASE,POINT2[] " "}
DECL PDAT PP_OLP9={VEL 100.0,ACC 100.0,APO_DIST 10.0,APO_MODE #CDIS}
DECL E6POS Xl040={X 430.074799,Y 1136.45398,Z -92.2810364,A 177.289993,B 20.8532009,C 89.6921234,S 2,T 10,E1 -5800.00293,E2 0.0,E3 0.0,E4 0.0,E5 0.0,E6 0.0}
DECL FDAT Fl045={TOOL_NO 4,BASE_NO 3,IPO_FRAME #BASE,POINT2[] " "}
DECL PDAT PP_OLP10={VEL 100.0,ACC 100.0,APO_DIST 10.0,APO_MODE #CDIS}
DECL E6POS Xl045={X 509.435303,Y 989.946777,Z 67.0658188,A 174.389099,B 74.1907578,C 83.2325134,S 2,T 43,E1 -5800.0,E2 0.0,E3 0.0,E4 0.0,E5 0.0,E6 0.0}
DECL FDAT Fl050={TOOL_NO 4,BASE_NO 3,IPO_FRAME #BASE,POINT2[] " "}
DECL PDAT PP_OLP11={VEL 100.0,ACC 100.0,APO_DIST 10.0,APO_MODE #CDIS}
DECL E6POS Xl050={X 518.755981,Y 1000.375,Z -62.166111,A -179.400894,B 74.3072433,C 88.9349213,S 2,T 11,E1 -5800.00293,E2 0.0,E3 0.0,E4 0.0,E5 0.0,E6 0.0}
DECL LDAT LL_OLP5={VEL 2.0,ACC 100.0,APO_DIST 0.0,APO_FAC 0.0,ORI_TYP #VAR,CIRC_TYP #BASE,JERK_FAC 50.0}
DECL LDAT LL_OLP6={VEL 2.0,ACC 100.0,APO_DIST 0.0,APO_FAC 0.0,ORI_TYP #VAR,CIRC_TYP #BASE,JERK_FAC 50.0}
DECL LDAT LL_OLP7={VEL 2.0,ACC 100.0,APO_DIST 0.0,APO_FAC 0.0,ORI_TYP #VAR,CIRC_TYP #BASE,JERK_FAC 50.0}
DECL LDAT LL_OLP8={VEL 2.0,ACC 100.0,APO_DIST 0.0,APO_FAC 0.0,ORI_TYP #VAR,CIRC_TYP #BASE,JERK_FAC 50.0}
DECL FDAT Fl055={TOOL_NO 4,BASE_NO 3,IPO_FRAME #BASE,POINT2[] " "}
DECL PDAT PP_OLP12={VEL 100.0,ACC 100.0,APO_DIST 20.0,APO_MODE #CDIS}
DECL E6POS Xl055={X 421.79361,Y 992.496399,Z -63.9221001,A 177.804596,B 74.2783737,C 86.1298599,S 2,T 11,E1 -5800.0,E2 0.0,E3 0.0,E4 0.0,E5 0.0,E6 0.0}
DECL FDAT Fl060={TOOL_NO 4,BASE_NO 3,IPO_FRAME #BASE,POINT2[] " "}
DECL PDAT PP_OLP13={VEL 100.0,ACC 100.0,APO_DIST 20.0,APO_MODE #CDIS}
DECL E6POS Xl060={X 685.309387,Y 1064.14905,Z 560.342224,A -176.427994,B -20.6658001,C 85.0904007,S 2,T 11,E1 -5800.0,E2 0.0,E3 0.0,E4 0.0,E5 0.0,E6 0.0}
DECL FDAT Fl065={TOOL_NO 4,BASE_NO 3,IPO_FRAME #BASE,POINT2[] " "}
DECL PDAT PP_OLP14={VEL 100.0,ACC 100.0,APO_DIST 0.0}
DECL E6POS Xl065={X 670.492004,Y 977.463989,Z 1154.84399,A -176.427994,B -20.6658001,C 85.0904007,S 2,T 11,E1 -5800.0,E2 0.0,E3 0.0,E4 0.0,E5 0.0,E6 0.0}
DECL FDAT Fl070={TOOL_NO 4,BASE_NO 3,IPO_FRAME #BASE,POINT2[] " "}
DECL PDAT PP_OLP15={VEL 100.0,ACC 100.0,APO_DIST 10.0,APO_MODE #CDIS}
DECL E6POS Xl070={X 663.247925,Y 988.811279,Z 1214.526,A -163.663605,B -54.7341385,C 79.5065613,S 2,T 11,E1 -5800.0,E2 0.0,E3 0.0,E4 0.0,E5 0.0,E6 0.0}
DECL FDAT FSWP_60_7780={TOOL_NO 4,BASE_NO 3,IPO_FRAME #BASE,POINT2[] " "}
DECL E6POS XSWP_60_7780={X 494.855408,Y 966.90741,Z 1255.66699,A -171.460602,B -55.4662704,C 81.8798828,S 2,T 11,E1 -5800.0,E2 0.0,E3 0.0,E4 0.0,E5 0.0,E6 0.0}
DECL LDAT LL_OLP9={VEL 2.0,ACC 100.0,APO_DIST 0.0,APO_FAC 0.0,ORI_TYP #VAR,CIRC_TYP #BASE,JERK_FAC 50.0}
DECL FDAT FSWP_60_7782={TOOL_NO 4,BASE_NO 3,IPO_FRAME #BASE,POINT2[] " "}
DECL E6POS XSWP_60_7782={X 519.43927,Y 965.740417,Z 1286.79602,A -175.917603,B -55.7446594,C 85.5283127,S 2,T 11,E1 -5800.0,E2 0.0,E3 0.0,E4 0.0,E5 0.0,E6 0.0}
DECL LDAT LL_OLP10={VEL 2.0,ACC 100.0,APO_DIST 0.0,APO_FAC 0.0,ORI_TYP #VAR,CIRC_TYP #BASE,JERK_FAC 50.0}
DECL FDAT FSWP_60_7784={TOOL_NO 4,BASE_NO 3,IPO_FRAME #BASE,POINT2[] " "}
DECL E6POS XSWP_60_7784={X 538.49408,Y 965.839417,Z 1300.89197,A -171.206802,B -55.4479485,C 81.6060562,S 2,T 11,E1 -5800.00391,E2 0.0,E3 0.0,E4 0.0,E5 0.0,E6 0.0}
DECL LDAT LL_OLP11={VEL 2.0,ACC 100.0,APO_DIST 0.0,APO_FAC 0.0,ORI_TYP #VAR,CIRC_TYP #BASE,JERK_FAC 50.0}
DECL FDAT Fl075={TOOL_NO 4,BASE_NO 3,IPO_FRAME #BASE,POINT2[] " "}
DECL PDAT PP_OLP16={VEL 100.0,ACC 100.0,APO_DIST 10.0,APO_MODE #CDIS}
DECL E6POS Xl075={X 588.503113,Y 965.342285,Z 1268.24805,A -167.772095,B -55.1350784,C 79.5641708,S 2,T 11,E1 -5800.00391,E2 0.0,E3 0.0,E4 0.0,E5 0.0,E6 0.0}
DECL FDAT Fl080={TOOL_NO 4,BASE_NO 3,IPO_FRAME #BASE,POINT2[] " "}
DECL PDAT PP_OLP17={VEL 100.0,ACC 100.0,APO_DIST 10.0,APO_MODE #CDIS}
DECL E6POS Xl080={X 668.778015,Y 962.935974,Z 1004.80701,A -176.427994,B -20.6658001,C 85.0904007,S 2,T 11,E1 -5800.0,E2 0.0,E3 0.0,E4 0.0,E5 0.0,E6 0.0}
DECL FDAT Fl085={TOOL_NO 4,BASE_NO 3,IPO_FRAME #BASE,POINT2[] " "}
DECL PDAT PP_OLP18={VEL 100.0,ACC 100.0,APO_DIST 10.0,APO_MODE #CDIS}
DECL E6POS Xl085={X 537.276428,Y 1134.94495,Z 884.519104,A -162.946899,B -49.510849,C 63.9570808,S 2,T 11,E1 -5800.00195,E2 0.0,E3 0.0,E4 0.0,E5 0.0,E6 0.0}
DECL FDAT Fl090={TOOL_NO 4,BASE_NO 3,IPO_FRAME #BASE,POINT2[] " "}
DECL PDAT PP_OLP19={VEL 100.0,ACC 100.0,APO_DIST 50.0,APO_MODE #CDIS}
DECL E6POS Xl090={X 1790.70703,Y 1260.84998,Z 125.791397,A -132.210602,B -34.5745392,C -9.67346478,S 2,T 3,E1 -4591.4458,E2 0.0,E3 0.0,E4 0.0,E5 0.0,E6 0.0}
DECL FDAT Fl095={TOOL_NO 4,BASE_NO 3,IPO_FRAME #BASE,POINT2[] " "}
DECL PDAT PP_OLP20={VEL 100.0,ACC 100.0,APO_DIST 50.0,APO_MODE #CDIS}
DECL E6POS Xl095={X 1756.96899,Y 1124.08203,Z 16.6684093,A -110.230598,B -29.0105209,C -48.4439507,S 2,T 35,E1 -4412.10791,E2 0.0,E3 0.0,E4 0.0,E5 0.0,E6 0.0}
DECL FDAT Fl100={TOOL_NO 4,BASE_NO 3,IPO_FRAME #BASE,POINT2[] " "}
DECL PDAT PP_OLP21={VEL 100.0,ACC 100.0,APO_DIST 50.0,APO_MODE #CDIS}
DECL E6POS Xl100={X 1639.66895,Y 657.687683,Z 111.432602,A -91.3977509,B -17.3471508,C -88.238327,S 2,T 35,E1 -4200.0,E2 0.0,E3 0.0,E4 0.0,E5 0.0,E6 0.0}
DECL FDAT Fl140={TOOL_NO 4,BASE_NO 3,IPO_FRAME #BASE,POINT2[] " "}
DECL E6POS Xl140={X 1629.84399,Y 680.869812,Z 97.8296585,A -89.2168503,B -16.9990692,C -88.7015076,S 2,T 35,E1 -4200.0,E2 0.0,E3 0.0,E4 0.0,E5 0.0,E6 0.0}
DECL FDAT Fl145={TOOL_NO 4,BASE_NO 3,IPO_FRAME #BASE,POINT2[] " "}
DECL E6POS Xl145={X 1630.71997,Y 616.697083,Z 117.462799,A -89.2169037,B -16.9996605,C -88.701889,S 2,T 35,E1 -4200.0,E2 0.0,E3 0.0,E4 0.0,E5 0.0,E6 0.0}
DECL LDAT LL_OLP20={VEL 1.0,ACC 100.0,APO_DIST 20.0,APO_FAC 0.0,ORI_TYP #VAR,CIRC_TYP #BASE,JERK_FAC 50.0}
DECL FDAT Fl150={TOOL_NO 4,BASE_NO 3,IPO_FRAME #BASE,POINT2[] " "}
DECL E6POS Xl150={X 1631.021,Y 603.029175,Z 116.371597,A -89.2170029,B -16.9997101,C -88.7019501,S 2,T 35,E1 -4200.0,E2 0.0,E3 0.0,E4 0.0,E5 0.0,E6 0.0}
DECL LDAT LL_OLP21={VEL 1.0,ACC 100.0,APO_DIST 20.0,APO_FAC 0.0,ORI_TYP #VAR,CIRC_TYP #BASE,JERK_FAC 50.0}
DECL FDAT FSWP_60_7532={TOOL_NO 4,BASE_NO 3,IPO_FRAME #BASE,POINT2[] " "}
DECL E6POS XSWP_60_7532={X 1637.67603,Y 599.048096,Z 124.444504,A -89.2175369,B -17.0010891,C -88.7023315,S 2,T 35,E1 -4200.0,E2 0.0,E3 0.0,E4 0.0,E5 0.0,E6 0.0}
DECL LDAT LL_OLP22={VEL 2.0,ACC 100.0,APO_DIST 0.0,APO_FAC 0.0,ORI_TYP #VAR,CIRC_TYP #BASE,JERK_FAC 50.0}
DECL FDAT Fl155={TOOL_NO 4,BASE_NO 3,IPO_FRAME #BASE,POINT2[] " "}
DECL E6POS Xl155={X 1628.73303,Y 598.014587,Z 120.842598,A -89.21698,B -16.9997005,C -88.7016068,S 2,T 35,E1 -4200.0,E2 0.0,E3 0.0,E4 0.0,E5 0.0,E6 0.0}
DECL LDAT LL_OLP23={VEL 1.0,ACC 100.0,APO_DIST 20.0,APO_FAC 0.0,ORI_TYP #VAR,CIRC_TYP #BASE,JERK_FAC 50.0}
DECL FDAT Fl160={TOOL_NO 4,BASE_NO 3,IPO_FRAME #BASE,POINT2[] " "}
DECL E6POS Xl160={X 1630.71997,Y 616.698181,Z 117.4655,A -89.2169037,B -16.9996395,C -88.7020035,S 2,T 35,E1 -4200.0,E2 0.0,E3 0.0,E4 0.0,E5 0.0,E6 0.0}
DECL LDAT LL_OLP24={VEL 1.0,ACC 100.0,APO_DIST 20.0,APO_FAC 0.0,ORI_TYP #VAR,CIRC_TYP #BASE,JERK_FAC 50.0}
DECL FDAT Fl180={TOOL_NO 4,BASE_NO 3,IPO_FRAME #BASE,POINT2[] " "}
DECL E6POS Xl180={X 1629.84302,Y 680.874878,Z 97.8408127,A -89.2169189,B -16.9996796,C -88.7018967,S 2,T 35,E1 -4200.0,E2 0.0,E3 0.0,E4 0.0,E5 0.0,E6 0.0}
DECL LDAT LL_OLP30={VEL 1.0,ACC 100.0,APO_DIST 20.0,APO_FAC 0.0,ORI_TYP #VAR,CIRC_TYP #BASE,JERK_FAC 50.0}
DECL FDAT Fl190={TOOL_NO 4,BASE_NO 3,IPO_FRAME #BASE,POINT2[] " "}
DECL E6POS Xl190={X 1634.81006,Y 709.458923,Z 104.760201,A -88.3470001,B -59.8070984,C -91.3890991,S 2,T 35,E1 -4200.0,E2 0.0,E3 0.0,E4 0.0,E5 0.0,E6 0.0}
DECL LDAT LL_OLP32={VEL 1.0,ACC 100.0,APO_DIST 20.0,APO_FAC 0.0,ORI_TYP #VAR,CIRC_TYP #BASE,JERK_FAC 50.0}
DECL FDAT FSWP_60_7524={TOOL_NO 4,BASE_NO 3,IPO_FRAME #BASE,POINT2[] " "}
DECL E6POS XSWP_60_7524={X 1640.896,Y 679.857422,Z 147.401093,A -88.7503967,B -48.775219,C -91.0600204,S 2,T 35,E1 -4200.0,E2 0.0,E3 0.0,E4 0.0,E5 0.0,E6 0.0}
DECL LDAT LL_OLP33={VEL 2.0,ACC 100.0,APO_DIST 0.0,APO_FAC 0.0,ORI_TYP #VAR,CIRC_TYP #BASE,JERK_FAC 50.0}
DECL FDAT FSWP_60_7522={TOOL_NO 4,BASE_NO 3,IPO_FRAME #BASE,POINT2[] " "}
DECL E6POS XSWP_60_7522={X 1639.95398,Y 722.280701,Z 146.387405,A -88.1218033,B -63.9261818,C -91.5929031,S 2,T 35,E1 -4200.0,E2 0.0,E3 0.0,E4 0.0,E5 0.0,E6 0.0}
DECL LDAT LL_OLP34={VEL 2.0,ACC 100.0,APO_DIST 0.0,APO_FAC 0.0,ORI_TYP #VAR,CIRC_TYP #BASE,JERK_FAC 50.0}
DECL FDAT FSWP_60_7518={TOOL_NO 4,BASE_NO 3,IPO_FRAME #BASE,POINT2[] " "}
DECL E6POS XSWP_60_7518={X 1640.18604,Y 777.721375,Z 142.4328,A -86.7086029,B -76.1517792,C -92.9305115,S 2,T 35,E1 -4199.99707,E2 0.0,E3 0.0,E4 0.0,E5 0.0,E6 0.0}
DECL LDAT LL_OLP36={VEL 2.0,ACC 100.0,APO_DIST 0.0,APO_FAC 0.0,ORI_TYP #VAR,CIRC_TYP #BASE,JERK_FAC 50.0}
DECL FDAT FSWP_60_7514={TOOL_NO 4,BASE_NO 3,IPO_FRAME #BASE,POINT2[] " "}
DECL E6POS XSWP_60_7514={X 1640.85498,Y 831.647278,Z 140.995804,A -74.860527,B -87.247139,C -104.708,S 2,T 35,E1 -4200.0,E2 0.0,E3 0.0,E4 0.0,E5 0.0,E6 0.0}
DECL LDAT LL_OLP38={VEL 2.0,ACC 100.0,APO_DIST 0.0,APO_FAC 0.0,ORI_TYP #VAR,CIRC_TYP #BASE,JERK_FAC 50.0}
DECL FDAT FSWP_60_7508={TOOL_NO 4,BASE_NO 3,IPO_FRAME #BASE,POINT2[] " "}
DECL E6POS XSWP_60_7508={X 1637.31702,Y 879.044678,Z 140.547806,A 72.4296112,B -87.7443314,C 108.035301,S 2,T 35,E1 -4200.0,E2 0.0,E3 0.0,E4 0.0,E5 0.0,E6 0.0}
DECL LDAT LL_OLP40={VEL 2.0,ACC 100.0,APO_DIST 0.0,APO_FAC 0.0,ORI_TYP #VAR,CIRC_TYP #BASE,JERK_FAC 50.0}
DECL FDAT FSWP_60_7510={TOOL_NO 4,BASE_NO 3,IPO_FRAME #BASE,POINT2[] " "}
DECL E6POS XSWP_60_7510={X 1640.40796,Y 926.516724,Z 139.793106,A 82.0300903,B -85.2440338,C 98.4500885,S 2,T 35,E1 -4200.0,E2 0.0,E3 0.0,E4 0.0,E5 0.0,E6 0.0}
DECL LDAT LL_OLP41={VEL 2.0,ACC 100.0,APO_DIST 0.0,APO_FAC 0.0,ORI_TYP #VAR,CIRC_TYP #BASE,JERK_FAC 50.0}
DECL FDAT FSWP_60_7512={TOOL_NO 4,BASE_NO 3,IPO_FRAME #BASE,POINT2[] " "}
DECL E6POS XSWP_60_7512={X 1635.64502,Y 969.374878,Z 139.662094,A 82.972023,B -84.638237,C 97.5117569,S 2,T 35,E1 -4200.0,E2 0.0,E3 0.0,E4 0.0,E5 0.0,E6 0.0}
DECL LDAT LL_OLP42={VEL 2.0,ACC 100.0,APO_DIST 0.0,APO_FAC 0.0,ORI_TYP #VAR,CIRC_TYP #BASE,JERK_FAC 50.0}
DECL FDAT Fl195={TOOL_NO 4,BASE_NO 3,IPO_FRAME #BASE,POINT2[] " "}
DECL PDAT PP_OLP28={VEL 100.0,ACC 100.0,APO_DIST 20.0,APO_MODE #CDIS}
DECL E6POS Xl195={X 1636.34094,Y 956.40863,Z 120.256897,A 90.7935867,B -75.187973,C 90.1105423,S 2,T 35,E1 -4200.0,E2 0.0,E3 0.0,E4 0.0,E5 0.0,E6 0.0}
DECL FDAT Fl200={TOOL_NO 4,BASE_NO 3,IPO_FRAME #BASE,POINT2[] " "}
DECL PDAT PP_OLP29={VEL 100.0,ACC 100.0,APO_DIST 20.0,APO_MODE #CDIS}
DECL E6POS Xl200={X 1642.09802,Y 1066.42505,Z 34.7488518,A 97.3658829,B -73.9743881,C 79.2817764,S 2,T 35,E1 -4200.0,E2 0.0,E3 0.0,E4 0.0,E5 0.0,E6 0.0}
DECL FDAT Fl210={TOOL_NO 4,BASE_NO 3,IPO_FRAME #BASE,POINT2[] " "}
DECL PDAT PP_OLP31={VEL 100.0,ACC 100.0,APO_DIST 20.0,APO_MODE #CDIS}
DECL E6POS Xl210={X 1646.71594,Y 1174.552,Z -11.3231497,A 149.347794,B -55.6305313,C 28.8826103,S 2,T 35,E1 -4200.06201,E2 0.0,E3 0.0,E4 0.0,E5 0.0,E6 0.0}
DECL FDAT Fl215={TOOL_NO 4,BASE_NO 3,IPO_FRAME #BASE,POINT2[] " "}
DECL PDAT PP_OLP32={VEL 100.0,ACC 100.0,APO_DIST 50.0,APO_MODE #CDIS}
DECL E6POS Xl215={X 1919.08704,Y 1695.06799,Z 259.654999,A 167.506897,B -6.48655319,C 38.056881,S 2,T 43,E1 -4304.58496,E2 0.0,E3 0.0,E4 0.0,E5 0.0,E6 0.0}
DECL BASIS_SUGG_T LAST_BASIS={POINT1[] "P0                      ",POINT2[] "P0                      ",CP_PARAMS[] "CPDAT0                  ",PTP_PARAMS[] "PDAT0                   ",CONT[] "                        ",CP_VEL[] "2.0                     ",PTP_VEL[] " 100                    ",SYNC_PARAMS[] "SYNCDAT                 ",SPL_NAME[] "S0                      "}
DECL E6POS XP1={X 339.203613,Y 946.779175,Z -220.366699,A -9.56965065,B -83.4578018,C -78.8764496,S 2,T 11,E1 -5800.0,E2 0.0,E3 0.0,E4 0.0,E5 0.0,E6 0.0}
DECL FDAT FP1={TOOL_NO 4,BASE_NO 3,IPO_FRAME #BASE,POINT2[] " ",TQ_STATE FALSE}
DECL PDAT PPDAT1={VEL 100.0,ACC 100.0,APO_DIST 20.0,APO_MODE #CDIS}
DECL E6POS XP2={X 365.644714,Y 943.723328,Z -200.357697,A 0.746322215,B -74.3037491,C -89.2692871,S 2,T 11,E1 -5800.0,E2 0.0,E3 0.0,E4 0.0,E5 0.0,E6 0.0}
DECL FDAT FP2={TOOL_NO 4,BASE_NO 3,IPO_FRAME #BASE,POINT2[] " ",TQ_STATE FALSE}
DECL PDAT PPDAT2={VEL 100.0,ACC 100.0,APO_DIST 20.0,APO_MODE #CDIS}
DECL E6POS XP3={X 370.62561,Y 946.708191,Z -192.170593,A 0.745761395,B -74.3037567,C -89.2687531,S 2,T 11,E1 -5800.0,E2 0.0,E3 0.0,E4 0.0,E5 0.0,E6 0.0}
DECL FDAT FP3={TOOL_NO 4,BASE_NO 3,IPO_FRAME #BASE,POINT2[] " ",TQ_STATE FALSE}
DECL PDAT PPDAT3={VEL 100.0,ACC 100.0,APO_DIST 20.0,APO_MODE #CDIS}
DECL SPOT_SUGG_T LAST_SPOT={GUN[] "1                       ",RETR_CMD[] "#OPN                    ",CHOISE[] "#FIRST                  ",CLO_TM[] "0                       ",PGNO1[] "1                       ",PRESS1[] "0                       ",PGNO2[] "1                       ",PRESS2[] "0                       ",SPOT_PARAMS[] "NORMAL                  "}
DECL E6POS XP13={X 1788.40601,Y 1032.55396,Z 1315.66699,A 179.958801,B -0.00576574123,C 81.505928,S 2,T 43,E1 -4799.99121,E2 0.0,E3 0.0,E4 0.0,E5 0.0,E6 0.0}
DECL FDAT FP13={TOOL_NO 4,BASE_NO 3,IPO_FRAME #BASE,POINT2[] " ",TQ_STATE FALSE}
DECL PDAT PPDAT11={VEL 100.0,ACC 100.0,APO_DIST 100.0}
DECL E6POS XSWP_60_9076={X 403.339111,Y 997.757202,Z -87.0384827,A 174.352997,B 74.194809,C 83.199791,S 2,T 11,E1 -5800.0,E2 0.0,E3 0.0,E4 0.0,E5 0.0,E6 0.0}
DECL FDAT FSWP_60_9076={TOOL_NO 4,BASE_NO 3,IPO_FRAME #BASE,POINT2[] " ",TQ_STATE FALSE}
DECL E6POS XSWP_60_9074={X 433.368805,Y 1000.33801,Z -101.3563,A 174.397003,B 74.1916122,C 83.2402267,S 2,T 11,E1 -5800.0,E2 0.0,E3 0.0,E4 0.0,E5 0.0,E6 0.0}
DECL FDAT FSWP_60_9074={TOOL_NO 4,BASE_NO 3,IPO_FRAME #BASE,POINT2[] " ",TQ_STATE FALSE}
DECL E6POS XSWP_60_9072={X 468.963287,Y 999.945129,Z -107.417198,A 174.389893,B 74.190979,C 83.2337036,S 2,T 11,E1 -5800.0,E2 0.0,E3 0.0,E4 0.0,E5 0.0,E6 0.0}
DECL FDAT FSWP_60_9072={TOOL_NO 4,BASE_NO 3,IPO_FRAME #BASE,POINT2[] " ",TQ_STATE FALSE}
DECL E6POS XSWP_60_9070={X 497.978088,Y 999.274902,Z -106.942902,A 174.397598,B 74.1919937,C 83.2398911,S 2,T 11,E1 -5800.00293,E2 0.0,E3 0.0,E4 0.0,E5 0.0,E6 0.0}
DECL FDAT FSWP_60_9070={TOOL_NO 4,BASE_NO 3,IPO_FRAME #BASE,POINT2[] " ",TQ_STATE FALSE}
DECL E6POS XSWP_60_9054={X 433.109589,Y 956.559326,Z -184.043198,A -0.126494899,B -82.8533096,C -88.4113083,S 2,T 11,E1 -5800.0,E2 0.0,E3 0.0,E4 0.0,E5 0.0,E6 0.0}
DECL FDAT FSWP_60_9054={TOOL_NO 4,BASE_NO 3,IPO_FRAME #BASE,POINT2[] " ",TQ_STATE FALSE}
DECL E6POS XSWP_60_9048={X 402.055695,Y 955.780579,Z -183.605194,A -4.06826591,B -87.937088,C -84.4787292,S 2,T 11,E1 -5800.0,E2 0.0,E3 0.0,E4 0.0,E5 0.0,E6 0.0}
DECL FDAT FSWP_60_9048={TOOL_NO 4,BASE_NO 3,IPO_FRAME #BASE,POINT2[] " ",TQ_STATE FALSE}
DECL E6POS XSWP_60_9050={X 370.621887,Y 955.240723,Z -184.882797,A -39.9076996,B -89.6957474,C -48.6436806,S 2,T 11,E1 -5800.0,E2 0.0,E3 0.0,E4 0.0,E5 0.0,E6 0.0}
DECL FDAT FSWP_60_9050={TOOL_NO 4,BASE_NO 3,IPO_FRAME #BASE,POINT2[] " ",TQ_STATE FALSE}
DECL E6POS XSWP_60_9052={X 337.679291,Y 956.125916,Z -189.675003,A -0.303649098,B -83.5875931,C -88.2352295,S 2,T 11,E1 -5800.0,E2 0.0,E3 0.0,E4 0.0,E5 0.0,E6 0.0}
DECL FDAT FSWP_60_9052={TOOL_NO 4,BASE_NO 3,IPO_FRAME #BASE,POINT2[] " ",TQ_STATE FALSE}
DECL E6POS XL091={X 1465.70105,Y 1457.42603,Z -47.5596504,A -139.776001,B -26.7611694,C 9.34067059,S 2,T 11,E1 -5055.68408,E2 0.0,E3 0.0,E4 0.0,E5 0.0,E6 0.0}
DECL FDAT Fl091={TOOL_NO 4,BASE_NO 3,IPO_FRAME #BASE,POINT2[] " ",TQ_STATE FALSE}
DECL PDAT PPDAT12={VEL 100.0,ACC 100.0,APO_DIST 50.0,APO_MODE #CDIS}
DECL LDAT LCPDAT3={VEL 2.0,ACC 100.0,APO_DIST 20.0,APO_FAC 50.0,AXIS_VEL 100.0,AXIS_ACC 100.0,ORI_TYP #VAR,CIRC_TYP #BASE,JERK_FAC 50.0,GEAR_JERK 50.0,EXAX_IGN 0}
DECL E6POS XP14={X 1811.60596,Y 1419.88696,Z 214.153595,A 158.230103,B -36.0415802,C 36.9010696,S 2,T 35,E1 -4264.92676,E2 0.0,E3 0.0,E4 0.0,E5 0.0,E6 0.0}
DECL FDAT FP14={TOOL_NO 4,BASE_NO 3,IPO_FRAME #BASE,POINT2[] " ",TQ_STATE FALSE}
DECL PDAT PPDAT13={VEL 100.0,ACC 100.0,APO_DIST 50.0,APO_MODE #CDIS}
DECL E6POS XP15={X 1763.83496,Y 1297.58801,Z 193.927002,A 151.769608,B -48.8652306,C 39.22855,S 2,T 35,E1 -4200.03711,E2 0.0,E3 0.0,E4 0.0,E5 0.0,E6 0.0}
DECL FDAT FP15={TOOL_NO 4,BASE_NO 3,IPO_FRAME #BASE,POINT2[] " ",TQ_STATE FALSE}
DECL PDAT PPDAT14={VEL 100.0,ACC 100.0,APO_DIST 50.0,APO_MODE #CDIS}
DECL PDAT PPDAT0={VEL 100.0,ACC 100.0,APO_DIST 100.0}
DECL E6POS XP0={X 6609.02393,Y 2724.13794,Z -373.295807,A 177.9729,B -20.0008602,C 0.623595595,S 2,T 2,E1 450.928497,E2 0.0,E3 0.0,E4 0.0,E5 0.0,E6 0.0}
DECL FDAT FP0={TOOL_NO 4,BASE_NO 3,IPO_FRAME #BASE,POINT2[] " ",TQ_STATE FALSE}
DECL PDAT PP_OLP2={VEL 100.0,ACC 100.0,APO_DIST 0.0}
DECL E6POS Xl005={X 3494.47412,Y 2838.10693,Z -263.893005,A -178.070496,B -0.250400007,C -0.44780001,S 2,T 2,E1 -3199.99805,E2 0.0,E3 0.0,E4 0.0,E5 0.0,E6 0.0}
DECL FDAT Fl005={TOOL_NO 4,BASE_NO 3,IPO_FRAME #BASE,POINT2[] " ",TQ_STATE FALSE}
DECL PDAT PPDAT4={VEL 100.0,ACC 100.0,APO_DIST 100.0}
DECL E6POS XP4={X 392.917511,Y 1131.21704,Z -209.6082,A -17.6624794,B -79.1884537,C -69.3067169,S 2,T 10,E1 -5800.0,E2 0.0,E3 0.0,E4 0.0,E5 0.0,E6 0.0}
DECL FDAT FP4={TOOL_NO 4,BASE_NO 3,IPO_FRAME #BASE,POINT2[] " ",TQ_STATE FALSE}
DECL PDAT PPDAT5={VEL 100.0,ACC 100.0,APO_DIST 50.0,APO_MODE #CDIS}
DECL E6POS XP5={X 580.025024,Y 1441.05298,Z -58.6644783,A -94.3374023,B -63.8539581,C -7.51724815,S 2,T 10,E1 -5286.26904,E2 0.0,E3 0.0,E4 0.0,E5 0.0,E6 0.0}
DECL FDAT FP5={TOOL_NO 4,BASE_NO 3,IPO_FRAME #BASE,POINT2[] " ",TQ_STATE FALSE}
DECL PDAT PP_OLP26={VEL 100.0,ACC 100.0,APO_DIST 20.0,APO_MODE #CDIS}
DECL E6POS Xl116={X 723.238892,Y 1953.323,Z -138.308594,A -173.140701,B -25.2844791,C 30.2326908,S 2,T 10,E1 -5014.13281,E2 0.0,E3 0.0,E4 0.0,E5 0.0,E6 0.0}
DECL FDAT Fl116={TOOL_NO 4,BASE_NO 3,IPO_FRAME #BASE,POINT2[] " "}
DECL PDAT PP_OLP25={VEL 100.0,ACC 100.0,APO_DIST 20.0,APO_MODE #CDIS}
DECL E6POS Xl120={X 3494.48291,Y 2838.10693,Z -263.893005,A -178.070496,B -0.250400007,C -0.44780001,S 2,T 2,E1 -3199.99805,E2 0.0,E3 0.0,E4 0.0,E5 0.0,E6 0.0}
DECL FDAT Fl120={TOOL_NO 4,BASE_NO 3,IPO_FRAME #BASE,POINT2[] " "}
DECL PDAT PPDAT6={VEL 100.0,ACC 100.0,APO_DIST 100.0}
DECL E6POS XP6={X 6613.13916,Y 2724.13208,Z -373.290894,A 177.972504,B -19.9948101,C 0.623847127,S 2,T 10,E1 199.999603,E2 0.0,E3 0.0,E4 0.0,E5 0.0,E6 0.0}
DECL FDAT FP6={TOOL_NO 4,BASE_NO 3,IPO_FRAME #BASE,POINT2[] " ",TQ_STATE FALSE}
DECL PDAT PP_OLP22={VEL 100.0,ACC 100.0,APO_DIST 50.0,APO_MODE #CDIS}
DECL E6POS Xl101={X 1798.83105,Y 494.3992,Z 111.142197,A -87.1523666,B -17.3469391,C -88.2307129,S 2,T 35,E1 -4200.0,E2 0.0,E3 0.0,E4 0.0,E5 0.0,E6 0.0}
DECL FDAT Fl101={TOOL_NO 4,BASE_NO 3,IPO_FRAME #BASE,POINT2[] " "}
DECL PDAT PP_OLP23={VEL 100.0,ACC 100.0,APO_DIST 50.0,APO_MODE #CDIS}
DECL E6POS Xl102={X 1892.25598,Y 275.513885,Z 134.641006,A 132.689697,B -64.2522507,C 43.5044098,S 2,T 35,E1 -4319.15576,E2 0.0,E3 0.0,E4 0.0,E5 0.0,E6 0.0}
DECL FDAT Fl102={TOOL_NO 4,BASE_NO 3,IPO_FRAME #BASE,POINT2[] " "}
DECL PDAT PP_OLP78={VEL 100.0,ACC 100.0,APO_DIST 100.0,APO_MODE #CDIS}
DECL E6POS Xl460={X 1629.78406,Y 621.88562,Z 89.3798523,A -16.0074291,B -89.2715988,C -163.541504,S 2,T 35,E1 -4200.0,E2 0.0,E3 0.0,E4 0.0,E5 0.0,E6 0.0}
DECL FDAT Fl460={TOOL_NO 4,BASE_NO 3,IPO_FRAME #BASE,POINT2[] " "}
DECL PDAT PP_OLP77={VEL 100.0,ACC 100.0,APO_DIST 100.0,APO_MODE #CDIS}
DECL E6POS Xl455={X 1721.48804,Y 606.746887,Z 91.6513672,A -16.0081902,B -89.2715988,C -163.540802,S 2,T 35,E1 -4200.0,E2 0.0,E3 0.0,E4 0.0,E5 0.0,E6 0.0}
DECL FDAT Fl455={TOOL_NO 4,BASE_NO 3,IPO_FRAME #BASE,POINT2[] " "}
DECL PDAT PP_OLP76={VEL 100.0,ACC 100.0,APO_DIST 100.0,APO_MODE #CDIS}
DECL E6POS Xl450={X 1737.15906,Y 324.549988,Z 146.149506,A -16.0210991,B -89.2717896,C -163.527893,S 2,T 35,E1 -4200.0,E2 0.0,E3 0.0,E4 0.0,E5 0.0,E6 0.0}
DECL FDAT Fl450={TOOL_NO 4,BASE_NO 3,IPO_FRAME #BASE,POINT2[] " "}
DECL PDAT PP_OLP75={VEL 100.0,ACC 100.0,APO_DIST 100.0,APO_MODE #CDIS}
DECL E6POS Xl445={X 1748.48096,Y 288.238892,Z 184.690399,A -139.888,B -85.6020432,C -38.2009392,S 2,T 35,E1 -4200.0,E2 0.0,E3 0.0,E4 0.0,E5 0.0,E6 0.0}
DECL FDAT Fl445={TOOL_NO 4,BASE_NO 3,IPO_FRAME #BASE,POINT2[] " "}
DECL PDAT PP_OLP79={VEL 100.0,ACC 100.0,APO_DIST 100.0,APO_MODE #CDIS}
DECL E6POS Xl446={X 1632.80896,Y 296.822906,Z 305.320099,A 90.9707336,B -75.1561737,C 90.3874435,S 2,T 35,E1 -4200.0,E2 0.0,E3 0.0,E4 0.0,E5 0.0,E6 0.0}
DECL FDAT Fl446={TOOL_NO 4,BASE_NO 3,IPO_FRAME #BASE,POINT2[] " "}
DECL LDAT LL_OLP25={VEL 2.0,ACC 100.0,APO_DIST 0.0,APO_FAC 0.0,ORI_TYP #VAR,CIRC_TYP #BASE,JERK_FAC 50.0}
DECL E6POS XSWP_60_7533={X 1635.72095,Y 595.326721,Z 120.626297,A -89.2177811,B -17.0006809,C -88.7020416,S 2,T 35,E1 -4200.0,E2 0.0,E3 0.0,E4 0.0,E5 0.0,E6 0.0}
DECL FDAT FSWP_60_7533={TOOL_NO 4,BASE_NO 3,IPO_FRAME #BASE,POINT2[] " "}
DECL E6POS XSWP_60_7536={X 1645.48596,Y 320.742004,Z 320.864014,A 88.9393311,B -65.1745682,C 91.6658401,S 2,T 35,E1 -4200.0,E2 0.0,E3 0.0,E4 0.0,E5 0.0,E6 0.0}
DECL FDAT FSWP_60_7536={TOOL_NO 4,BASE_NO 3,IPO_FRAME #BASE,POINT2[] " ",TQ_STATE FALSE}
DECL LDAT LL_OLP35={VEL 2.0,ACC 100.0,APO_DIST 0.0,APO_FAC 0.0,ORI_TYP #VAR,CIRC_TYP #BASE,JERK_FAC 50.0}
DECL E6POS XSWP_60_7537={X 1638.25403,Y 320.97171,Z 322.661194,A 87.8068237,B -75.168457,C 92.7347336,S 2,T 35,E1 -4200.0,E2 0.0,E3 0.0,E4 0.0,E5 0.0,E6 0.0}
DECL FDAT FSWP_60_7537={TOOL_NO 4,BASE_NO 3,IPO_FRAME #BASE,POINT2[] " "}
DECL LDAT LL_OLP37={VEL 2.0,ACC 100.0,APO_DIST 0.0,APO_FAC 0.0,ORI_TYP #VAR,CIRC_TYP #BASE,JERK_FAC 50.0}
DECL E6POS XSWP_60_7538={X 1641.15698,Y 279.335999,Z 349.428589,A 87.8128967,B -75.1694031,C 92.7301025,S 2,T 35,E1 -4200.0,E2 0.0,E3 0.0,E4 0.0,E5 0.0,E6 0.0}
DECL FDAT FSWP_60_7538={TOOL_NO 4,BASE_NO 3,IPO_FRAME #BASE,POINT2[] " "}
DECL LDAT LL_OLP39={VEL 2.0,ACC 100.0,APO_DIST 0.0,APO_FAC 0.0,ORI_TYP #VAR,CIRC_TYP #BASE,JERK_FAC 50.0}
DECL E6POS XSWP_60_7540={X 1641.53601,Y 227.337006,Z 352.581512,A 81.5671616,B -85.4863434,C 98.9122162,S 2,T 35,E1 -4200.0,E2 0.0,E3 0.0,E4 0.0,E5 0.0,E6 0.0}
DECL FDAT FSWP_60_7540={TOOL_NO 4,BASE_NO 3,IPO_FRAME #BASE,POINT2[] " "}
DECL PDAT PP_OLP80={VEL 100.0,ACC 100.0,APO_DIST 100.0,APO_MODE #CDIS}
DECL E6POS Xl447={X 1643.63696,Y 251.093002,Z 292.402802,A -117.209702,B -86.9634705,C -62.9117317,S 2,T 35,E1 -4200.0,E2 0.0,E3 0.0,E4 0.0,E5 0.0,E6 0.0}
DECL FDAT Fl447={TOOL_NO 4,BASE_NO 3,IPO_FRAME #BASE,POINT2[] " "}
DECL PDAT PP_OLP81={VEL 100.0,ACC 100.0,APO_DIST 100.0,APO_MODE #CDIS}
DECL E6POS Xl451={X 1936.89905,Y 193.901794,Z 111.412903,A -146.987793,B -66.6449966,C -26.90625,S 2,T 35,E1 -4200.0,E2 0.0,E3 0.0,E4 0.0,E5 0.0,E6 0.0}
DECL FDAT Fl451={TOOL_NO 4,BASE_NO 3,IPO_FRAME #BASE,POINT2[] " "}
DECL PDAT PP_OLP24={VEL 100.0,ACC 100.0,APO_DIST 50.0,APO_MODE #CDIS}
DECL E6POS Xl103={X 1874.203,Y 1166.26099,Z 95.5545425,A -97.5552673,B -13.6891499,C -46.9793892,S 2,T 3,E1 -4200.06201,E2 0.0,E3 0.0,E4 0.0,E5 0.0,E6 0.0}
DECL FDAT Fl103={TOOL_NO 4,BASE_NO 3,IPO_FRAME #BASE,POINT2[] " "}
DECL PDAT PP_OLP27={VEL 100.0,ACC 100.0,APO_DIST 50.0,APO_MODE #CDIS}
DECL E6POS Xl104={X 1892.25598,Y 275.513885,Z 134.641006,A 132.689697,B -64.2522507,C 43.5044098,S 2,T 35,E1 -4319.15576,E2 0.0,E3 0.0,E4 0.0,E5 0.0,E6 0.0}
DECL FDAT Fl104={TOOL_NO 4,BASE_NO 3,IPO_FRAME #BASE,POINT2[] " "}
DECL PDAT PP_OLP30={VEL 100.0,ACC 100.0,APO_DIST 50.0,APO_MODE #CDIS}
DECL E6POS Xl105={X 1967.51404,Y 1081.35498,Z 131.5672,A 164.735504,B -57.1573601,C 10.8218603,S 2,T 35,E1 -4200.06201,E2 0.0,E3 0.0,E4 0.0,E5 0.0,E6 0.0}
DECL FDAT Fl105={TOOL_NO 4,BASE_NO 3,IPO_FRAME #BASE,POINT2[] " "}
DECL PDAT Pvmax={VEL 100.0,ACC 100.0,APO_DIST 100.0}
DECL LDAT Lvmax={VEL 2.0,ACC 100.0,APO_DIST 100.0,APO_FAC 50.0,AXIS_VEL 100.0,AXIS_ACC 100.0,ORI_TYP #VAR,CIRC_TYP #BASE,JERK_FAC 50.0,GEAR_JERK 50.0,EXAX_IGN 0}
DECL PDAT PPDAT7={VEL 100.0,ACC 100.0,APO_DIST 100.0}
DECL PDAT Pfin={VEL 100.0,ACC 100.0,APO_DIST 20.0,APO_MODE #CDIS}
DECL PDAT Pxlarge={VEL 100.0,ACC 100.0,APO_DIST 500.0,APO_MODE #CDIS}
DECL PDAT Plarge={VEL 100.0,ACC 100.0,APO_DIST 200.0,APO_MODE #CDIS}
DECL PDAT Pmedium={VEL 100.0,ACC 100.0,APO_DIST 100.0,APO_MODE #CDIS}
DECL PDAT Psmall={VEL 100.0,ACC 100.0,APO_DIST 50.0,APO_MODE #CDIS}
DECL PDAT Pxxlarge={VEL 100.0,ACC 100.0,APO_DIST 1000.0,APO_MODE #CDIS}
ENDDAT
